Yaskawa INFORM job: DEMO_ROOF_SIDE_0625_3PAINT_12.JBI

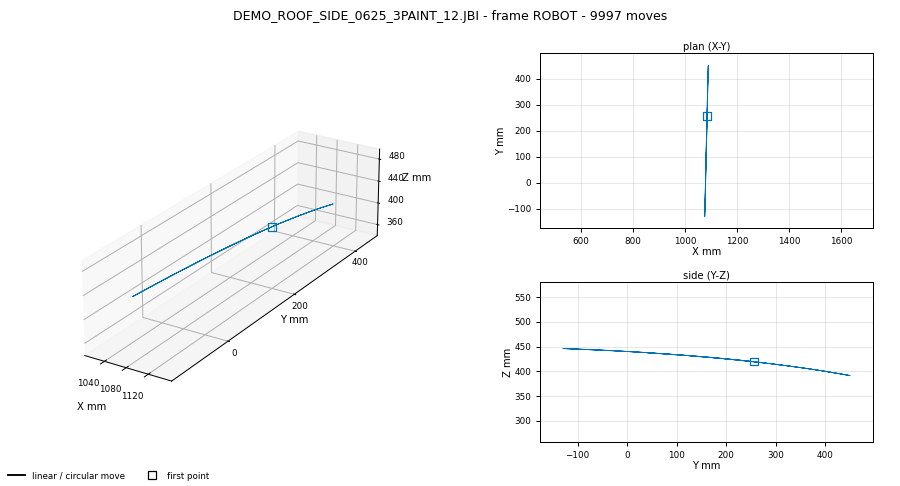
[picture p0: tool path of DEMO_ROOF_SIDE_0625_3PAINT_12.JBI in frame ROBOT, 9997 of 9997 moves have a stored position in this frame; points joined in program order, loops and branches not executed]
/JOB
//NAME DEMO_ROOF_SIDE_0625_3PAINT12
//POS
///NPOS 9997,0,0,0,0,0
///TOOL 0
///USER 0
///POSTYPE ROBOT
///RECTAN
///RCONF 1,0,0,0,0,0,0,0,0,0,0,0,0,0,0,0,0,0,0,0,0,0,0,0
C00000=1085.651,255.676,419.931,175.989,23.066,153.710
C00001=1085.645,255.428,419.959,175.986,23.063,153.710
C00002=1085.640,255.179,419.986,175.983,23.060,153.710
C00003=1085.635,254.931,420.014,175.981,23.057,153.709
C00004=1085.628,254.682,420.041,175.978,23.054,153.709
C00005=1085.623,254.434,420.069,175.975,23.051,153.709
C00006=1085.617,254.186,420.096,175.973,23.048,153.709
C00007=1085.611,253.937,420.124,175.970,23.045,153.708
C00008=1085.606,253.689,420.151,175.967,23.041,153.708
C00009=1085.600,253.441,420.179,175.965,23.039,153.708
C00010=1085.595,253.192,420.206,175.962,23.035,153.707
C00011=1085.589,252.943,420.233,175.959,23.032,153.707
C00012=1085.584,252.695,420.261,175.956,23.029,153.707
C00013=1085.578,252.446,420.287,175.953,23.026,153.707
C00014=1085.573,252.198,420.315,175.951,23.024,153.706
C00015=1085.567,251.950,420.342,175.948,23.020,153.706
C00016=1085.561,251.701,420.370,175.945,23.017,153.706
C00017=1085.555,251.453,420.397,175.943,23.014,153.705
C00018=1085.550,251.204,420.424,175.940,23.011,153.705
C00019=1085.544,250.956,420.451,175.937,23.008,153.705
C00020=1085.539,250.707,420.478,175.935,23.005,153.705
C00021=1085.532,250.459,420.506,175.932,23.002,153.704
C00022=1085.527,250.210,420.533,175.929,22.999,153.704
C00023=1085.519,249.831,420.575,175.925,22.995,153.704
C00024=1085.511,249.453,420.616,175.921,22.990,153.703
C00025=1085.502,249.074,420.657,175.917,22.986,153.703
C00026=1085.494,248.695,420.698,175.912,22.980,153.702
C00027=1085.488,248.447,420.725,175.910,22.978,153.702
C00028=1085.483,248.199,420.753,175.907,22.974,153.702
C00029=1085.477,247.950,420.780,175.905,22.972,153.702
C00030=1085.471,247.702,420.806,175.902,22.969,153.701
C00031=1085.466,247.453,420.834,175.899,22.965,153.701
C00032=1085.460,247.204,420.861,175.897,22.963,153.701
C00033=1085.455,246.956,420.888,175.894,22.959,153.700
C00034=1085.449,246.707,420.915,175.892,22.957,153.700
C00035=1085.443,246.459,420.941,175.889,22.954,153.700
C00036=1085.438,246.210,420.968,175.886,22.951,153.700
C00037=1085.432,245.962,420.995,175.883,22.948,153.699
C00038=1085.427,245.713,421.022,175.880,22.945,153.699
C00039=1085.421,245.465,421.048,175.878,22.942,153.699
C00040=1085.416,245.216,421.076,175.875,22.939,153.699
C00041=1085.409,244.967,421.103,175.872,22.936,153.698
C00042=1085.404,244.719,421.129,175.870,22.933,153.698
C00043=1085.398,244.471,421.156,175.867,22.930,153.698
C00044=1085.393,244.222,421.183,175.865,22.927,153.698
C00045=1085.387,243.974,421.210,175.862,22.924,153.697
C00046=1085.381,243.725,421.236,175.859,22.921,153.697
C00047=1085.376,243.477,421.263,175.857,22.918,153.697
C00048=1085.370,243.228,421.290,175.854,22.915,153.696
C00049=1085.365,242.980,421.317,175.851,22.912,153.696
C00050=1085.359,242.731,421.343,175.848,22.909,153.696
C00051=1085.353,242.482,421.370,175.845,22.906,153.696
C00052=1085.348,242.234,421.396,175.843,22.903,153.695
C00053=1085.342,241.986,421.423,175.840,22.900,153.695
C00054=1085.336,241.737,421.450,175.838,22.897,153.695
C00055=1085.330,241.489,421.476,175.835,22.894,153.695
C00056=1085.325,241.240,421.502,175.833,22.892,153.694
C00057=1085.319,240.992,421.529,175.830,22.889,153.694
C00058=1085.313,240.743,421.556,175.827,22.885,153.694
C00059=1085.307,240.494,421.582,175.824,22.883,153.694
C00060=1085.302,240.245,421.608,175.821,22.880,153.693
C00061=1085.296,239.997,421.635,175.819,22.877,153.693
C00062=1085.291,239.748,421.662,175.816,22.874,153.693
C00063=1085.285,239.500,421.688,175.814,22.871,153.693
C00064=1085.279,239.251,421.714,175.811,22.868,153.692
C00065=1085.273,239.003,421.741,175.809,22.865,153.692
C00066=1085.267,238.754,421.767,175.806,22.863,153.692
C00067=1085.262,238.506,421.793,175.803,22.859,153.692
C00068=1085.257,238.258,421.820,175.800,22.857,153.691
C00069=1085.251,238.009,421.846,175.797,22.853,153.691
C00070=1085.245,237.761,421.872,175.795,22.851,153.691
C00071=1085.240,237.512,421.898,175.792,22.848,153.691
C00072=1085.234,237.263,421.925,175.790,22.845,153.690
C00073=1085.228,237.015,421.952,175.787,22.842,153.690
C00074=1085.223,236.766,421.977,175.785,22.839,153.690
C00075=1085.214,236.380,422.019,175.780,22.834,153.690
C00076=1085.205,235.995,422.059,175.777,22.830,153.689
C00077=1085.196,235.609,422.100,175.772,22.825,153.689
C00078=1085.188,235.224,422.140,175.768,22.821,153.688
C00079=1085.182,234.975,422.166,175.765,22.818,153.688
C00080=1085.177,234.726,422.192,175.763,22.815,153.688
C00081=1085.171,234.478,422.219,175.760,22.812,153.688
C00082=1085.165,234.229,422.244,175.758,22.809,153.687
C00083=1085.159,233.981,422.271,175.755,22.806,153.687
C00084=1085.154,233.732,422.297,175.753,22.804,153.687
C00085=1085.149,233.484,422.323,175.750,22.800,153.687
C00086=1085.143,233.235,422.349,175.748,22.798,153.686
C00087=1085.138,232.986,422.375,175.745,22.794,153.686
C00088=1085.131,232.738,422.400,175.742,22.791,153.686
C00089=1085.126,232.489,422.427,175.739,22.789,153.686
C00090=1085.120,232.240,422.453,175.736,22.786,153.685
C00091=1085.115,231.991,422.479,175.734,22.783,153.685
C00092=1085.109,231.744,422.505,175.731,22.780,153.685
C00093=1085.103,231.495,422.531,175.729,22.777,153.684
C00094=1085.098,231.246,422.557,175.726,22.774,153.684
C00095=1085.092,230.997,422.582,175.724,22.771,153.684
C00096=1085.086,230.749,422.609,175.721,22.768,153.684
C00097=1085.081,230.501,422.634,175.719,22.765,153.683
C00098=1085.076,230.252,422.660,175.716,22.762,153.683
C00099=1085.069,230.003,422.685,175.713,22.760,153.683
C00100=1085.064,229.754,422.711,175.710,22.757,153.683
C00101=1085.058,229.506,422.738,175.708,22.754,153.682
C00102=1085.052,229.257,422.763,175.705,22.751,153.682
C00103=1085.047,229.009,422.789,175.703,22.748,153.682
C00104=1085.041,228.760,422.814,175.700,22.745,153.682
C00105=1085.035,228.511,422.840,175.698,22.742,153.681
C00106=1085.030,228.262,422.866,175.696,22.740,153.681
C00107=1085.024,228.013,422.891,175.692,22.737,153.681
C00108=1085.019,227.765,422.917,175.690,22.734,153.681
C00109=1085.013,227.516,422.942,175.687,22.731,153.681
C00110=1085.007,227.267,422.968,175.685,22.728,153.680
C00111=1085.001,227.019,422.994,175.682,22.725,153.680
C00112=1084.996,226.771,423.020,175.680,22.722,153.680
C00113=1084.990,226.522,423.045,175.677,22.719,153.680
C00114=1084.984,226.273,423.071,175.675,22.716,153.679
C00115=1084.979,226.024,423.097,175.672,22.714,153.679
C00116=1084.973,225.777,423.122,175.669,22.711,153.679
C00117=1084.968,225.528,423.148,175.666,22.708,153.679
C00118=1084.962,225.278,423.173,175.664,22.705,153.678
C00119=1084.957,225.030,423.198,175.661,22.702,153.678
C00120=1084.951,224.781,423.223,175.659,22.699,153.678
C00121=1084.945,224.532,423.249,175.656,22.696,153.678
C00122=1084.939,224.284,423.275,175.654,22.693,153.677
C00123=1084.934,224.035,423.300,175.652,22.691,153.677
C00124=1084.928,223.787,423.326,175.649,22.688,153.677
C00125=1084.923,223.538,423.351,175.646,22.685,153.677
C00126=1084.917,223.290,423.377,175.643,22.682,153.676
C00127=1084.908,222.895,423.417,175.640,22.678,153.676
C00128=1084.900,222.501,423.457,175.635,22.673,153.675
C00129=1084.890,222.107,423.497,175.632,22.668,153.675
C00130=1084.882,221.713,423.537,175.627,22.663,153.675
C00131=1084.875,221.464,423.562,175.625,22.661,153.675
C00132=1084.870,221.215,423.588,175.622,22.658,153.674
C00133=1084.865,220.967,423.612,175.620,22.655,153.674
C00134=1084.858,220.718,423.637,175.618,22.652,153.674
C00135=1084.853,220.469,423.663,175.615,22.649,153.674
C00136=1084.847,220.221,423.688,175.612,22.647,153.673
C00137=1084.841,219.972,423.713,175.609,22.643,153.673
C00138=1084.836,219.724,423.738,175.607,22.641,153.673
C00139=1084.830,219.475,423.764,175.604,22.638,153.673
C00140=1084.824,219.226,423.789,175.602,22.635,153.672
C00141=1084.819,218.978,423.813,175.600,22.632,153.672
C00142=1084.813,218.729,423.839,175.597,22.630,153.672
C00143=1084.808,218.480,423.864,175.595,22.627,153.672
C00144=1084.802,218.231,423.889,175.592,22.623,153.671
C00145=1084.796,217.982,423.914,175.590,22.621,153.671
C00146=1084.790,217.734,423.939,175.586,22.618,153.671
C00147=1084.784,217.485,423.963,175.584,22.615,153.671
C00148=1084.780,217.237,423.989,175.582,22.612,153.670
C00149=1084.773,216.988,424.014,175.579,22.609,153.670
C00150=1084.768,216.739,424.038,175.577,22.607,153.670
C00151=1084.762,216.491,424.064,175.574,22.604,153.670
C00152=1084.757,216.242,424.088,175.572,22.601,153.669
C00153=1084.751,215.993,424.114,175.570,22.598,153.669
C00154=1084.746,215.745,424.138,175.566,22.595,153.669
C00155=1084.740,215.496,424.164,175.564,22.592,153.669
C00156=1084.734,215.247,424.188,175.561,22.589,153.668
C00157=1084.728,214.998,424.212,175.559,22.586,153.668
C00158=1084.724,214.750,424.238,175.557,22.584,153.668
C00159=1084.718,214.500,424.263,175.554,22.581,153.668
C00160=1084.712,214.252,424.288,175.552,22.578,153.667
C00161=1084.706,214.003,424.312,175.549,22.575,153.667
C00162=1084.701,213.755,424.336,175.547,22.572,153.667
C00163=1084.695,213.506,424.362,175.544,22.570,153.667
C00164=1084.689,213.257,424.386,175.541,22.566,153.666
C00165=1084.683,213.009,424.411,175.539,22.564,153.666
C00166=1084.679,212.760,424.436,175.536,22.560,153.666
C00167=1084.673,212.510,424.461,175.534,22.558,153.666
C00168=1084.667,212.262,424.485,175.532,22.555,153.665
C00169=1084.661,212.013,424.510,175.529,22.552,153.665
C00170=1084.656,211.765,424.535,175.527,22.549,153.665
C00171=1084.651,211.516,424.559,175.524,22.546,153.665
C00172=1084.644,211.267,424.584,175.522,22.544,153.664
C00173=1084.639,211.019,424.609,175.520,22.541,153.664
C00174=1084.633,210.770,424.633,175.517,22.538,153.664
C00175=1084.628,210.521,424.657,175.514,22.535,153.664
C00176=1084.622,210.272,424.682,175.512,22.532,153.663
C00177=1084.616,210.024,424.706,175.509,22.529,153.663
C00178=1084.610,209.775,424.731,175.507,22.526,153.663
C00179=1084.602,209.385,424.769,175.503,22.522,153.663
C00180=1084.592,208.995,424.808,175.499,22.518,153.662
C00181=1084.584,208.604,424.846,175.495,22.513,153.662
C00182=1084.575,208.214,424.884,175.492,22.509,153.661
C00183=1084.552,207.186,424.984,175.406,22.464,153.664
C00184=1084.547,206.937,425.007,175.403,22.462,153.664
C00185=1084.540,206.688,425.031,175.401,22.460,153.664
C00186=1084.535,206.439,425.056,175.398,22.458,153.664
C00187=1084.530,206.190,425.080,175.396,22.457,153.664
C00188=1084.524,205.941,425.103,175.393,22.455,153.664
C00189=1084.519,205.693,425.127,175.391,22.453,153.664
C00190=1084.512,205.444,425.151,175.387,22.451,153.664
C00191=1084.507,205.195,425.175,175.385,22.448,153.664
C00192=1084.502,204.946,425.199,175.383,22.447,153.664
C00193=1084.496,204.698,425.222,175.380,22.445,153.664
C00194=1084.491,204.449,425.246,175.378,22.443,153.664
C00195=1084.485,204.200,425.270,175.375,22.441,153.664
C00196=1084.479,203.952,425.294,175.373,22.439,153.664
C00197=1084.474,203.702,425.318,175.370,22.437,153.664
C00198=1084.468,203.454,425.342,175.367,22.435,153.664
C00199=1084.463,203.204,425.365,175.365,22.433,153.664
C00200=1084.457,202.956,425.389,175.362,22.431,153.664
C00201=1084.452,202.707,425.412,175.360,22.429,153.664
C00202=1084.446,202.458,425.437,175.357,22.428,153.664
C00203=1084.441,202.209,425.459,175.355,22.426,153.664
C00204=1084.434,201.960,425.483,175.352,22.424,153.664
C00205=1084.429,201.711,425.507,175.349,22.422,153.664
C00206=1084.423,201.463,425.531,175.347,22.420,153.664
C00207=1084.418,201.214,425.554,175.344,22.418,153.664
C00208=1084.412,200.965,425.578,175.342,22.416,153.664
C00209=1084.406,200.717,425.601,175.339,22.414,153.664
C00210=1084.401,200.468,425.625,175.337,22.413,153.664
C00211=1084.395,200.218,425.648,175.334,22.411,153.664
C00212=1084.389,199.970,425.672,175.332,22.409,153.664
C00213=1084.384,199.721,425.696,175.329,22.407,153.664
C00214=1084.378,199.473,425.719,175.327,22.405,153.664
C00215=1084.372,199.224,425.742,175.323,22.403,153.664
C00216=1084.367,198.974,425.766,175.321,22.401,153.664
C00217=1084.361,198.726,425.789,175.319,22.400,153.664
C00218=1084.355,198.477,425.812,175.316,22.398,153.664
C00219=1084.350,198.228,425.836,175.314,22.396,153.664
C00220=1084.344,197.980,425.860,175.311,22.394,153.664
C00221=1084.338,197.731,425.882,175.309,22.392,153.664
C00222=1084.333,197.481,425.906,175.306,22.390,153.663
C00223=1084.327,197.233,425.930,175.304,22.389,153.663
C00224=1084.321,196.984,425.953,175.301,22.387,153.663
C00225=1084.316,196.735,425.977,175.299,22.385,153.663
C00226=1084.310,196.486,426.000,175.296,22.383,153.663
C00227=1084.304,196.237,426.023,175.293,22.381,153.663
C00228=1084.299,195.988,426.047,175.291,22.379,153.663
C00229=1084.293,195.739,426.070,175.288,22.377,153.663
C00230=1084.287,195.491,426.093,175.286,22.375,153.663
C00231=1084.282,195.242,426.116,175.283,22.373,153.663
C00232=1084.277,194.993,426.140,175.281,22.371,153.663
C00233=1084.271,194.744,426.163,175.278,22.370,153.663
C00234=1084.265,194.495,426.186,175.276,22.368,153.663
C00235=1084.259,194.247,426.209,175.273,22.366,153.663
C00236=1084.254,193.998,426.233,175.271,22.364,153.663
C00237=1084.248,193.749,426.256,175.268,22.362,153.663
C00238=1084.243,193.500,426.279,175.266,22.361,153.663
C00239=1084.237,193.251,426.302,175.264,22.359,153.663
C00240=1084.232,193.002,426.325,175.261,22.356,153.663
C00241=1084.226,192.753,426.348,175.259,22.355,153.663
C00242=1084.221,192.505,426.371,175.256,22.353,153.663
C00243=1084.215,192.256,426.394,175.254,22.351,153.663
C00244=1084.209,191.977,426.420,175.251,22.349,153.663
C00245=1084.203,191.699,426.446,175.248,22.347,153.663
C00246=1084.197,191.420,426.472,175.245,22.344,153.663
C00247=1084.190,191.142,426.498,175.242,22.342,153.663
C00248=1084.185,190.893,426.521,175.240,22.341,153.663
C00249=1084.180,190.644,426.544,175.238,22.339,153.663
C00250=1084.174,190.395,426.567,175.235,22.337,153.663
C00251=1084.168,190.146,426.590,175.233,22.335,153.663
C00252=1084.162,189.897,426.613,175.230,22.333,153.663
C00253=1084.157,189.648,426.636,175.228,22.331,153.663
C00254=1084.152,189.400,426.659,175.225,22.329,153.663
C00255=1084.147,189.151,426.682,175.223,22.327,153.662
C00256=1084.141,188.902,426.705,175.220,22.326,153.662
C00257=1084.135,188.653,426.728,175.218,22.323,153.662
C00258=1084.129,188.404,426.751,175.216,22.321,153.662
C00259=1084.125,188.154,426.774,175.213,22.320,153.662
C00260=1084.120,187.906,426.796,175.211,22.318,153.662
C00261=1084.114,187.657,426.819,175.208,22.316,153.662
C00262=1084.108,187.408,426.842,175.206,22.314,153.662
C00263=1084.102,187.159,426.865,175.204,22.312,153.662
C00264=1084.097,186.910,426.888,175.201,22.310,153.662
C00265=1084.092,186.662,426.911,175.199,22.308,153.662
C00266=1084.087,186.412,426.933,175.196,22.306,153.662
C00267=1084.081,186.163,426.956,175.194,22.304,153.662
C00268=1084.075,185.915,426.979,175.191,22.302,153.662
C00269=1084.070,185.666,427.002,175.189,22.300,153.662
C00270=1084.065,185.418,427.025,175.187,22.299,153.662
C00271=1084.059,185.168,427.047,175.184,22.296,153.662
C00272=1084.053,184.919,427.070,175.182,22.295,153.662
C00273=1084.048,184.670,427.093,175.179,22.293,153.662
C00274=1084.042,184.421,427.116,175.177,22.291,153.662
C00275=1084.036,184.172,427.138,175.174,22.289,153.662
C00276=1084.031,183.924,427.160,175.172,22.287,153.662
C00277=1084.025,183.675,427.183,175.169,22.285,153.662
C00278=1084.019,183.426,427.206,175.167,22.284,153.662
C00279=1084.014,183.177,427.228,175.165,22.282,153.662
C00280=1084.007,182.928,427.251,175.162,22.280,153.662
C00281=1084.002,182.679,427.274,175.160,22.278,153.662
C00282=1083.996,182.430,427.296,175.157,22.276,153.662
C00283=1083.991,182.181,427.318,175.155,22.275,153.662
C00284=1083.985,181.933,427.341,175.152,22.273,153.661
C00285=1083.979,181.683,427.363,175.150,22.271,153.661
C00286=1083.973,181.434,427.386,175.147,22.269,153.661
C00287=1083.967,181.185,427.408,175.145,22.267,153.661
C00288=1083.961,180.936,427.430,175.142,22.265,153.661
C00289=1083.956,180.688,427.453,175.141,22.264,153.661
C00290=1083.951,180.439,427.475,175.138,22.262,153.661
C00291=1083.944,180.190,427.498,175.136,22.260,153.661
C00292=1083.939,179.940,427.520,175.133,22.259,153.661
C00293=1083.933,179.692,427.543,175.131,22.257,153.661
C00294=1083.928,179.443,427.564,175.129,22.254,153.661
C00295=1083.922,179.194,427.587,175.126,22.253,153.661
C00296=1083.917,178.945,427.609,175.124,22.251,153.661
C00297=1083.910,178.696,427.632,175.121,22.249,153.661
C00298=1083.905,178.447,427.653,175.119,22.247,153.661
C00299=1083.900,178.198,427.676,175.116,22.245,153.661
C00300=1083.893,177.949,427.698,175.114,22.244,153.661
C00301=1083.888,177.700,427.721,175.111,22.242,153.661
C00302=1083.883,177.451,427.743,175.109,22.240,153.661
C00303=1083.876,177.203,427.765,175.106,22.238,153.661
C00304=1083.871,176.953,427.787,175.105,22.236,153.661
C00305=1083.866,176.705,427.809,175.103,22.234,153.661
C00306=1083.860,176.456,427.832,175.100,22.233,153.661
C00307=1083.854,176.206,427.854,175.098,22.231,153.661
C00308=1083.848,175.928,427.879,175.095,22.229,153.661
C00309=1083.841,175.649,427.904,175.092,22.226,153.661
C00310=1083.836,175.370,427.929,175.090,22.224,153.661
C00311=1083.830,175.091,427.953,175.087,22.223,153.661
C00312=1083.823,174.842,427.975,175.085,22.221,153.661
C00313=1083.818,174.593,427.998,175.082,22.218,153.661
C00314=1083.813,174.344,428.020,175.080,22.217,153.660
C00315=1083.807,174.095,428.041,175.078,22.215,153.660
C00316=1083.801,173.846,428.064,175.075,22.213,153.660
C00317=1083.795,173.598,428.086,175.073,22.211,153.660
C00318=1083.790,173.348,428.108,175.070,22.209,153.660
C00319=1083.785,173.099,428.130,175.069,22.207,153.660
C00320=1083.779,172.851,428.152,175.066,22.206,153.660
C00321=1083.773,172.601,428.174,175.064,22.204,153.660
C00322=1083.768,172.353,428.196,175.061,22.202,153.660
C00323=1083.762,172.103,428.218,175.059,22.200,153.660
C00324=1083.757,171.854,428.240,175.057,22.198,153.660
C00325=1083.751,171.606,428.262,175.054,22.196,153.660
C00326=1083.745,171.356,428.284,175.052,22.194,153.660
C00327=1083.740,171.108,428.306,175.049,22.192,153.660
C00328=1083.735,170.858,428.328,175.048,22.190,153.660
C00329=1083.729,170.610,428.349,175.045,22.189,153.660
C00330=1083.724,170.360,428.371,175.043,22.187,153.660
C00331=1083.717,170.112,428.394,175.041,22.185,153.660
C00332=1083.712,169.863,428.415,175.038,22.183,153.660
C00333=1083.706,169.614,428.437,175.036,22.181,153.660
C00334=1083.701,169.365,428.459,175.033,22.179,153.660
C00335=1083.696,169.115,428.481,175.031,22.177,153.659
C00336=1083.690,168.867,428.502,175.029,22.175,153.659
C00337=1083.685,168.617,428.525,175.027,22.174,153.659
C00338=1083.679,168.369,428.546,175.025,22.172,153.659
C00339=1083.674,168.119,428.568,175.022,22.169,153.659
C00340=1083.668,167.871,428.589,175.020,22.168,153.659
C00341=1083.663,167.621,428.612,175.017,22.166,153.659
C00342=1083.657,167.373,428.633,175.015,22.163,153.659
C00343=1083.652,167.123,428.655,175.014,22.162,153.659
C00344=1083.646,166.875,428.676,175.011,22.160,153.659
C00345=1083.641,166.625,428.699,175.009,22.158,153.659
C00346=1083.635,166.377,428.720,175.006,22.156,153.659
C00347=1083.630,166.127,428.742,175.004,22.154,153.659
C00348=1083.624,165.879,428.763,175.002,22.152,153.659
C00349=1083.620,165.630,428.785,174.999,22.150,153.659
C00350=1083.613,165.381,428.807,174.998,22.149,153.659
C00351=1083.609,165.132,428.829,174.995,22.146,153.658
C00352=1083.602,164.883,428.850,174.993,22.145,153.658
C00353=1083.597,164.634,428.872,174.990,22.143,153.658
C00354=1083.591,164.385,428.894,174.988,22.140,153.658
C00355=1083.586,164.136,428.915,174.986,22.139,153.658
C00356=1083.581,163.887,428.937,174.984,22.137,153.658
C00357=1083.575,163.638,428.959,174.982,22.135,153.658
C00358=1083.570,163.389,428.980,174.979,22.133,153.658
C00359=1083.564,163.140,429.002,174.977,22.131,153.658
C00360=1083.559,162.891,429.023,174.975,22.129,153.658
C00361=1083.554,162.642,429.045,174.972,22.127,153.658
C00362=1083.548,162.393,429.066,174.971,22.125,153.658
C00363=1083.543,162.144,429.088,174.968,22.123,153.658
C00364=1083.538,161.895,429.109,174.966,22.121,153.658
C00365=1083.532,161.646,429.131,174.964,22.119,153.658
C00366=1083.527,161.397,429.152,174.961,22.117,153.657
C00367=1083.520,161.148,429.174,174.959,22.115,153.657
C00368=1083.515,160.899,429.194,174.957,22.114,153.657
C00369=1083.509,160.650,429.216,174.955,22.112,153.657
C00370=1083.504,160.401,429.238,174.953,22.109,153.657
C00371=1083.499,160.152,429.259,174.950,22.108,153.657
C00372=1083.492,159.872,429.283,174.948,22.106,153.657
C00373=1083.486,159.593,429.306,174.945,22.103,153.657
C00374=1083.480,159.314,429.330,174.943,22.102,153.657
C00375=1083.473,159.034,429.355,174.941,22.099,153.657
C00376=1083.468,158.785,429.375,174.938,22.097,153.657
C00377=1083.462,158.537,429.397,174.936,22.096,153.657
C00378=1083.456,158.288,429.418,174.934,22.093,153.657
C00379=1083.451,158.038,429.439,174.931,22.091,153.657
C00380=1083.445,157.789,429.461,174.930,22.090,153.657
C00381=1083.439,157.541,429.482,174.927,22.088,153.657
C00382=1083.435,157.291,429.503,174.925,22.086,153.657
C00383=1083.428,157.042,429.525,174.922,22.084,153.657
C00384=1083.423,156.793,429.545,174.920,22.082,153.656
C00385=1083.418,156.545,429.566,174.919,22.080,153.656
C00386=1083.411,156.295,429.588,174.916,22.079,153.656
C00387=1083.406,156.046,429.609,174.914,22.076,153.656
C00388=1083.401,155.798,429.630,174.911,22.074,153.656
C00389=1083.395,155.548,429.651,174.910,22.072,153.656
C00390=1083.389,155.299,429.672,174.908,22.071,153.656
C00391=1083.383,155.050,429.693,174.905,22.069,153.656
C00392=1083.378,154.801,429.714,174.903,22.066,153.656
C00393=1083.372,154.552,429.735,174.900,22.065,153.656
C00394=1083.366,154.303,429.756,174.899,22.063,153.656
C00395=1083.361,154.054,429.777,174.897,22.061,153.656
C00396=1083.355,153.805,429.798,174.894,22.059,153.656
C00397=1083.350,153.556,429.819,174.892,22.057,153.656
C00398=1083.344,153.307,429.840,174.890,22.055,153.655
C00399=1083.339,153.058,429.861,174.888,22.054,153.655
C00400=1083.333,152.809,429.882,174.885,22.052,153.655
C00401=1083.327,152.559,429.903,174.883,22.049,153.655
C00402=1083.322,152.310,429.924,174.882,22.048,153.655
C00403=1083.317,152.062,429.945,174.879,22.046,153.655
C00404=1083.311,151.812,429.966,174.877,22.044,153.655
C00405=1083.305,151.563,429.987,174.874,22.042,153.655
C00406=1083.300,151.314,430.008,174.873,22.040,153.655
C00407=1083.295,151.065,430.028,174.871,22.038,153.655
C00408=1083.288,150.816,430.050,174.868,22.036,153.655
C00409=1083.282,150.567,430.070,174.866,22.034,153.655
C00410=1083.277,150.318,430.090,174.864,22.033,153.655
C00411=1083.272,150.069,430.112,174.862,22.030,153.655
C00412=1083.266,149.820,430.133,174.860,22.029,153.654
C00413=1083.261,149.570,430.153,174.857,22.026,153.654
C00414=1083.255,149.322,430.175,174.856,22.025,153.654
C00415=1083.250,149.073,430.195,174.853,22.022,153.654
C00416=1083.244,148.823,430.216,174.851,22.021,153.654
C00417=1083.238,148.574,430.236,174.849,22.019,153.654
C00418=1083.232,148.326,430.257,174.847,22.017,153.654
C00419=1083.227,148.077,430.278,174.845,22.015,153.654
C00420=1083.221,147.827,430.299,174.842,22.013,153.654
C00421=1083.216,147.578,430.319,174.840,22.011,153.654
C00422=1083.210,147.329,430.340,174.838,22.010,153.654
C00423=1083.204,147.080,430.360,174.836,22.007,153.654
C00424=1083.199,146.830,430.381,174.834,22.005,153.654
C00425=1083.193,146.581,430.402,174.832,22.003,153.653
C00426=1083.187,146.333,430.422,174.830,22.002,153.653
C00427=1083.182,146.083,430.442,174.827,22.000,153.653
C00428=1083.176,145.835,430.464,174.825,21.997,153.653
C00429=1083.171,145.585,430.485,174.824,21.996,153.653
C00430=1083.165,145.336,430.505,174.821,21.994,153.653
C00431=1083.159,145.087,430.525,174.819,21.992,153.653
C00432=1083.154,144.838,430.546,174.817,21.990,153.653
C00433=1083.148,144.589,430.566,174.815,21.988,153.653
C00434=1083.142,144.339,430.587,174.813,21.986,153.653
C00435=1083.137,144.090,430.607,174.810,21.984,153.653
C00436=1083.131,143.811,430.630,174.808,21.982,153.653
C00437=1083.124,143.532,430.653,174.806,21.980,153.653
C00438=1083.119,143.252,430.676,174.803,21.977,153.652
C00439=1083.112,142.973,430.699,174.801,21.975,153.652
C00440=1083.107,142.724,430.719,174.799,21.973,153.652
C00441=1083.100,142.474,430.740,174.797,21.971,153.652
C00442=1083.095,142.225,430.760,174.795,21.970,153.652
C00443=1083.089,141.976,430.782,174.793,21.967,153.652
C00444=1083.083,141.728,430.802,174.791,21.966,153.652
C00445=1083.078,141.478,430.821,174.789,21.963,153.652
C00446=1083.073,141.229,430.842,174.786,21.962,153.652
C00447=1083.067,140.980,430.862,174.785,21.960,153.652
C00448=1083.062,140.731,430.882,174.783,21.958,153.652
C00449=1083.056,140.482,430.902,174.780,21.956,153.651
C00450=1083.050,140.232,430.923,174.779,21.954,153.651
C00451=1083.045,139.983,430.944,174.776,21.952,153.651
C00452=1083.039,139.734,430.964,174.774,21.950,153.651
C00453=1083.034,139.485,430.984,174.772,21.948,153.651
C00454=1083.028,139.236,431.004,174.770,21.946,153.651
C00455=1083.022,138.987,431.025,174.768,21.944,153.651
C00456=1083.016,138.738,431.045,174.766,21.942,153.651
C00457=1083.011,138.489,431.065,174.764,21.940,153.651
C00458=1083.005,138.240,431.085,174.762,21.938,153.651
C00459=1083.000,137.991,431.105,174.759,21.936,153.651
C00460=1082.994,137.741,431.125,174.758,21.935,153.651
C00461=1082.988,137.492,431.146,174.756,21.932,153.650
C00462=1082.982,137.243,431.166,174.753,21.930,153.650
C00463=1082.977,136.994,431.187,174.752,21.928,153.650
C00464=1082.971,136.745,431.206,174.750,21.926,153.650
C00465=1082.966,136.496,431.226,174.747,21.924,153.650
C00466=1082.960,136.247,431.246,174.746,21.922,153.650
C00467=1082.954,135.998,431.266,174.743,21.921,153.650
C00468=1082.949,135.749,431.287,174.741,21.918,153.650
C00469=1082.943,135.499,431.306,174.739,21.917,153.650
C00470=1082.938,135.250,431.327,174.737,21.914,153.650
C00471=1082.932,135.001,431.347,174.735,21.913,153.650
C00472=1082.927,134.752,431.367,174.733,21.911,153.649
C00473=1082.921,134.503,431.386,174.731,21.908,153.649
C00474=1082.916,134.254,431.407,174.729,21.906,153.649
C00475=1082.910,134.005,431.427,174.727,21.905,153.649
C00476=1082.904,133.755,431.446,174.725,21.903,153.649
C00477=1082.899,133.506,431.467,174.723,21.900,153.649
C00478=1082.893,133.258,431.487,174.721,21.898,153.649
C00479=1082.888,133.008,431.506,174.719,21.897,153.649
C00480=1082.882,132.759,431.526,174.717,21.894,153.649
C00481=1082.876,132.510,431.546,174.715,21.893,153.649
C00482=1082.871,132.260,431.566,174.713,21.891,153.648
C00483=1082.865,132.012,431.586,174.711,21.888,153.648
C00484=1082.859,131.763,431.606,174.709,21.887,153.648
C00485=1082.853,131.513,431.625,174.707,21.884,153.648
C00486=1082.848,131.264,431.646,174.705,21.883,153.648
C00487=1082.842,131.015,431.665,174.703,21.881,153.648
C00488=1082.836,130.766,431.685,174.700,21.879,153.648
C00489=1082.830,130.517,431.705,174.699,21.877,153.648
C00490=1082.825,130.268,431.724,174.697,21.875,153.648
C00491=1082.819,130.019,431.745,174.694,21.873,153.648
C00492=1082.814,129.769,431.764,174.693,21.871,153.647
C00493=1082.808,129.520,431.784,174.691,21.869,153.647
C00494=1082.802,129.271,431.803,174.688,21.867,153.647
C00495=1082.796,129.022,431.823,174.687,21.865,153.647
C00496=1082.790,128.773,431.843,174.685,21.863,153.647
C00497=1082.785,128.524,431.863,174.683,21.861,153.647
C00498=1082.779,128.274,431.882,174.681,21.859,153.647
C00499=1082.773,128.025,431.902,174.678,21.857,153.647
C00500=1082.767,127.745,431.924,174.676,21.855,153.647
C00501=1082.760,127.466,431.946,174.674,21.853,153.647
C00502=1082.754,127.186,431.969,174.672,21.851,153.646
C00503=1082.748,126.906,431.991,174.670,21.848,153.646
C00504=1082.742,126.657,432.010,174.668,21.846,153.646
C00505=1082.736,126.408,432.030,174.665,21.844,153.646
C00506=1082.731,126.159,432.049,174.664,21.842,153.646
C00507=1082.725,125.909,432.068,174.662,21.840,153.646
C00508=1082.719,125.661,432.088,174.660,21.838,153.646
C00509=1082.713,125.411,432.108,174.658,21.837,153.646
C00510=1082.708,125.163,432.127,174.656,21.834,153.646
C00511=1082.703,124.913,432.147,174.654,21.832,153.645
C00512=1082.697,124.664,432.166,174.652,21.831,153.645
C00513=1082.691,124.415,432.186,174.650,21.828,153.645
C00514=1082.685,124.166,432.205,174.648,21.826,153.645
C00515=1082.680,123.916,432.225,174.646,21.824,153.645
C00516=1082.674,123.667,432.245,174.644,21.822,153.645
C00517=1082.668,123.418,432.264,174.642,21.820,153.645
C00518=1082.662,123.168,432.283,174.640,21.818,153.645
C00519=1082.657,122.920,432.302,174.638,21.816,153.645
C00520=1082.651,122.671,432.322,174.636,21.814,153.644
C00521=1082.646,122.422,432.341,174.635,21.812,153.644
C00522=1082.641,122.172,432.361,174.632,21.810,153.644
C00523=1082.635,121.923,432.381,174.630,21.808,153.644
C00524=1082.629,121.674,432.400,174.629,21.806,153.644
C00525=1082.624,121.425,432.419,174.626,21.804,153.644
C00526=1082.618,121.175,432.438,174.625,21.802,153.644
C00527=1082.613,120.926,432.458,174.623,21.800,153.644
C00528=1082.607,120.677,432.478,174.620,21.798,153.643
C00529=1082.601,120.428,432.497,174.619,21.796,153.643
C00530=1082.596,120.179,432.516,174.617,21.794,153.643
C00531=1082.590,119.930,432.535,174.615,21.792,153.643
C00532=1082.584,119.680,432.554,174.613,21.789,153.643
C00533=1082.578,119.431,432.574,174.612,21.788,153.643
C00534=1082.573,119.182,432.593,174.609,21.785,153.643
C00535=1082.568,118.933,432.612,174.607,21.783,153.643
C00536=1082.562,118.684,432.632,174.606,21.781,153.642
C00537=1082.556,118.434,432.651,174.603,21.779,153.642
C00538=1082.551,118.185,432.670,174.602,21.777,153.642
C00539=1082.546,117.936,432.689,174.600,21.775,153.642
C00540=1082.540,117.687,432.708,174.597,21.773,153.642
C00541=1082.534,117.437,432.727,174.596,21.771,153.642
C00542=1082.528,117.188,432.747,174.594,21.769,153.642
C00543=1082.523,116.940,432.766,174.592,21.767,153.642
C00544=1082.517,116.690,432.785,174.590,21.764,153.641
C00545=1082.512,116.441,432.805,174.589,21.762,153.641
C00546=1082.507,116.192,432.824,174.586,21.761,153.641
C00547=1082.501,115.943,432.843,174.584,21.758,153.641
C00548=1082.495,115.693,432.862,174.583,21.756,153.641
C00549=1082.490,115.444,432.881,174.580,21.754,153.641
C00550=1082.484,115.195,432.900,174.579,21.752,153.641
C00551=1082.479,114.946,432.919,174.577,21.750,153.640
C00552=1082.473,114.696,432.939,174.575,21.748,153.640
C00553=1082.468,114.447,432.958,174.573,21.745,153.640
C00554=1082.462,114.198,432.977,174.572,21.744,153.640
C00555=1082.456,113.949,432.995,174.569,21.742,153.640
C00556=1082.450,113.699,433.015,174.567,21.739,153.640
C00557=1082.445,113.451,433.034,174.566,21.737,153.640
C00558=1082.440,113.201,433.052,174.564,21.735,153.640
C00559=1082.434,112.951,433.071,174.562,21.734,153.639
C00560=1082.428,112.703,433.090,174.560,21.731,153.639
C00561=1082.423,112.453,433.109,174.558,21.729,153.639
C00562=1082.417,112.204,433.128,174.556,21.727,153.639
C00563=1082.411,111.955,433.147,174.555,21.725,153.639
C00564=1082.405,111.676,433.168,174.553,21.723,153.639
C00565=1082.398,111.395,433.189,174.550,21.720,153.639
C00566=1082.392,111.116,433.210,174.548,21.718,153.638
C00567=1082.385,110.837,433.232,174.546,21.716,153.638
C00568=1082.380,110.587,433.250,174.544,21.714,153.638
C00569=1082.375,110.338,433.269,174.542,21.712,153.638
C00570=1082.368,110.089,433.288,174.541,21.710,153.638
C00571=1082.363,109.839,433.307,174.538,21.708,153.638
C00572=1082.357,109.590,433.326,174.536,21.705,153.638
C00573=1082.351,109.341,433.344,174.535,21.703,153.637
C00574=1082.346,109.092,433.363,174.533,21.701,153.637
C00575=1082.340,108.842,433.382,174.531,21.699,153.637
C00576=1082.334,108.594,433.401,174.529,21.697,153.637
C00577=1082.329,108.344,433.419,174.527,21.695,153.637
C00578=1082.322,108.095,433.438,174.525,21.693,153.637
C00579=1082.317,107.846,433.457,174.524,21.691,153.637
C00580=1082.312,107.596,433.476,174.522,21.689,153.637
C00581=1082.306,107.347,433.493,174.520,21.687,153.636
C00582=1082.300,107.098,433.513,174.518,21.685,153.636
C00583=1082.295,106.848,433.532,174.516,21.683,153.636
C00584=1082.289,106.599,433.550,174.514,21.680,153.636
C00585=1082.284,106.350,433.569,174.513,21.679,153.636
C00586=1082.277,106.101,433.587,174.511,21.676,153.636
C00587=1082.272,105.852,433.606,174.508,21.674,153.636
C00588=1082.267,105.602,433.625,174.507,21.672,153.635
C00589=1082.261,105.354,433.643,174.505,21.669,153.635
C00590=1082.255,105.104,433.662,174.503,21.668,153.635
C00591=1082.249,104.854,433.680,174.501,21.666,153.635
C00592=1082.244,104.606,433.699,174.500,21.664,153.635
C00593=1082.238,104.356,433.717,174.497,21.661,153.635
C00594=1082.233,104.107,433.736,174.496,21.659,153.635
C00595=1082.227,103.858,433.755,174.494,21.657,153.634
C00596=1082.221,103.608,433.773,174.492,21.655,153.634
C00597=1082.216,103.359,433.792,174.490,21.653,153.634
C00598=1082.210,103.110,433.810,174.489,21.651,153.634
C00599=1082.205,102.861,433.829,174.487,21.649,153.634
C00600=1082.199,102.611,433.847,174.485,21.647,153.634
C00601=1082.193,102.362,433.866,174.483,21.644,153.634
C00602=1082.187,102.113,433.884,174.482,21.642,153.633
C00603=1082.182,101.864,433.902,174.479,21.640,153.633
C00604=1082.177,101.614,433.921,174.478,21.638,153.633
C00605=1082.171,101.365,433.939,174.476,21.636,153.633
C00606=1082.166,101.115,433.958,174.475,21.634,153.633
C00607=1082.160,100.867,433.976,174.472,21.631,153.633
C00608=1082.154,100.617,433.994,174.471,21.629,153.632
C00609=1082.148,100.368,434.013,174.469,21.627,153.632
C00610=1082.143,100.119,434.031,174.467,21.625,153.632
C00611=1082.136,99.870,434.049,174.465,21.623,153.632
C00612=1082.131,99.620,434.068,174.464,21.621,153.632
C00613=1082.125,99.371,434.086,174.461,21.619,153.632
C00614=1082.119,99.122,434.104,174.460,21.617,153.632
C00615=1082.114,98.873,434.123,174.458,21.615,153.631
C00616=1082.108,98.624,434.141,174.456,21.613,153.631
C00617=1082.102,98.374,434.159,174.454,21.610,153.631
C00618=1082.096,98.125,434.178,174.453,21.608,153.631
C00619=1082.091,97.875,434.195,174.451,21.606,153.631
C00620=1082.085,97.626,434.213,174.449,21.604,153.631
C00621=1082.080,97.377,434.232,174.447,21.602,153.631
C00622=1082.074,97.127,434.250,174.446,21.600,153.630
C00623=1082.068,96.879,434.268,174.443,21.597,153.630
C00624=1082.062,96.629,434.287,174.442,21.596,153.630
C00625=1082.057,96.380,434.305,174.440,21.593,153.630
C00626=1082.050,96.131,434.323,174.438,21.591,153.630
C00627=1082.046,95.881,434.341,174.436,21.589,153.630
C00628=1082.039,95.602,434.361,174.435,21.587,153.629
C00629=1082.032,95.322,434.382,174.433,21.585,153.629
C00630=1082.026,95.042,434.402,174.431,21.582,153.629
C00631=1082.020,94.763,434.422,174.428,21.579,153.629
C00632=1082.015,94.514,434.440,174.427,21.577,153.629
C00633=1082.009,94.265,434.459,174.425,21.575,153.629
C00634=1082.003,94.015,434.476,174.423,21.573,153.628
C00635=1081.997,93.766,434.494,174.421,21.571,153.628
C00636=1081.992,93.516,434.513,174.420,21.569,153.628
C00637=1081.986,93.267,434.531,174.418,21.566,153.628
C00638=1081.980,93.018,434.549,174.416,21.564,153.628
C00639=1081.975,92.769,434.567,174.414,21.562,153.628
C00640=1081.969,92.519,434.585,174.413,21.560,153.627
C00641=1081.964,92.270,434.602,174.411,21.558,153.627
C00642=1081.957,92.021,434.621,174.409,21.556,153.627
C00643=1081.953,91.772,434.639,174.408,21.553,153.627
C00644=1081.947,91.523,434.657,174.406,21.551,153.627
C00645=1081.941,91.273,434.675,174.404,21.549,153.627
C00646=1081.935,91.024,434.692,174.402,21.547,153.626
C00647=1081.929,90.774,434.710,174.401,21.545,153.626
C00648=1081.924,90.525,434.728,174.399,21.542,153.626
C00649=1081.918,90.276,434.747,174.397,21.540,153.626
C00650=1081.913,90.027,434.765,174.395,21.538,153.626
C00651=1081.907,89.778,434.782,174.394,21.536,153.626
C00652=1081.901,89.528,434.800,174.391,21.534,153.625
C00653=1081.895,89.279,434.818,174.390,21.532,153.625
C00654=1081.889,89.029,434.836,174.388,21.529,153.625
C00655=1081.884,88.780,434.853,174.386,21.527,153.625
C00656=1081.878,88.531,434.871,174.385,21.526,153.625
C00657=1081.872,88.281,434.889,174.383,21.523,153.625
C00658=1081.867,88.032,434.906,174.382,21.521,153.625
C00659=1081.860,87.782,434.924,174.379,21.519,153.624
C00660=1081.855,87.533,434.942,174.378,21.517,153.624
C00661=1081.849,87.284,434.959,174.376,21.515,153.624
C00662=1081.843,87.035,434.977,174.374,21.513,153.624
C00663=1081.838,86.786,434.995,174.372,21.510,153.624
C00664=1081.832,86.536,435.013,174.371,21.508,153.624
C00665=1081.826,86.287,435.030,174.370,21.506,153.623
C00666=1081.821,86.038,435.048,174.367,21.503,153.623
C00667=1081.815,85.788,435.066,174.366,21.502,153.623
C00668=1081.809,85.539,435.083,174.364,21.499,153.623
C00669=1081.803,85.290,435.101,174.363,21.497,153.623
C00670=1081.797,85.040,435.119,174.360,21.495,153.623
C00671=1081.792,84.791,435.136,174.359,21.493,153.622
C00672=1081.786,84.542,435.154,174.357,21.491,153.622
C00673=1081.780,84.292,435.172,174.355,21.489,153.622
C00674=1081.775,84.043,435.189,174.354,21.487,153.622
C00675=1081.769,83.794,435.207,174.352,21.484,153.622
C00676=1081.764,83.545,435.224,174.351,21.482,153.621
C00677=1081.758,83.295,435.242,174.348,21.479,153.621
C00678=1081.752,83.046,435.259,174.347,21.477,153.621
C00679=1081.747,82.797,435.277,174.345,21.475,153.621
C00680=1081.741,82.547,435.295,174.344,21.473,153.621
C00681=1081.735,82.298,435.312,174.341,21.471,153.621
C00682=1081.730,82.049,435.330,174.340,21.468,153.620
C00683=1081.724,81.799,435.347,174.339,21.466,153.620
C00684=1081.718,81.550,435.365,174.337,21.464,153.620
C00685=1081.713,81.300,435.382,174.335,21.462,153.620
C00686=1081.707,81.051,435.400,174.333,21.460,153.620
C00687=1081.702,80.802,435.418,174.332,21.458,153.620
C00688=1081.696,80.552,435.435,174.330,21.455,153.619
C00689=1081.690,80.303,435.452,174.328,21.453,153.619
C00690=1081.684,80.054,435.469,174.327,21.451,153.619
C00691=1081.679,79.805,435.487,174.325,21.449,153.619
C00692=1081.673,79.525,435.507,174.323,21.446,153.619
C00693=1081.666,79.246,435.526,174.321,21.444,153.618
C00694=1081.660,78.966,435.545,174.319,21.441,153.618
C00695=1081.653,78.687,435.565,174.317,21.438,153.618
C00696=1081.648,78.437,435.582,174.316,21.437,153.618
C00697=1081.642,78.187,435.600,174.314,21.434,153.618
C00698=1081.636,77.938,435.618,174.312,21.432,153.617
C00699=1081.630,77.689,435.634,174.311,21.430,153.617
C00700=1081.625,77.440,435.651,174.309,21.427,153.617
C00701=1081.619,77.190,435.669,174.308,21.425,153.617
C00702=1081.614,76.941,435.686,174.305,21.423,153.617
C00703=1081.607,76.692,435.703,174.304,21.421,153.617
C00704=1081.602,76.443,435.721,174.303,21.419,153.616
C00705=1081.597,76.193,435.738,174.301,21.416,153.616
C00706=1081.590,75.944,435.755,174.299,21.414,153.616
C00707=1081.584,75.695,435.772,174.297,21.412,153.616
C00708=1081.579,75.445,435.789,174.296,21.410,153.616
C00709=1081.574,75.196,435.807,174.294,21.408,153.615
C00710=1081.567,74.946,435.823,174.292,21.406,153.615
C00711=1081.561,74.697,435.841,174.291,21.403,153.615
C00712=1081.556,74.448,435.859,174.289,21.401,153.615
C00713=1081.550,74.198,435.875,174.287,21.399,153.615
C00714=1081.544,73.949,435.892,174.285,21.396,153.615
C00715=1081.539,73.700,435.909,174.284,21.395,153.614
C00716=1081.533,73.450,435.927,174.283,21.392,153.614
C00717=1081.527,73.201,435.943,174.281,21.390,153.614
C00718=1081.522,72.952,435.961,174.279,21.388,153.614
C00719=1081.516,72.702,435.978,174.277,21.385,153.614
C00720=1081.510,72.453,435.995,174.276,21.383,153.613
C00721=1081.505,72.204,436.012,174.275,21.381,153.613
C00722=1081.499,71.954,436.030,174.272,21.379,153.613
C00723=1081.493,71.704,436.046,174.271,21.377,153.613
C00724=1081.487,71.455,436.063,174.269,21.374,153.613
C00725=1081.482,71.206,436.080,174.268,21.372,153.612
C00726=1081.476,70.957,436.097,174.266,21.370,153.612
C00727=1081.471,70.707,436.114,174.264,21.367,153.612
C00728=1081.464,70.459,436.131,174.263,21.365,153.612
C00729=1081.459,70.208,436.148,174.261,21.363,153.612
C00730=1081.453,69.959,436.166,174.259,21.361,153.612
C00731=1081.447,69.710,436.182,174.258,21.359,153.611
C00732=1081.442,69.460,436.199,174.256,21.356,153.611
C00733=1081.436,69.212,436.216,174.255,21.354,153.611
C00734=1081.430,68.962,436.233,174.253,21.352,153.611
C00735=1081.424,68.713,436.250,174.251,21.349,153.611
C00736=1081.419,68.463,436.267,174.250,21.348,153.610
C00737=1081.414,68.214,436.283,174.248,21.345,153.610
C00738=1081.407,67.964,436.301,174.246,21.343,153.610
C00739=1081.402,67.715,436.318,174.245,21.341,153.610
C00740=1081.396,67.465,436.334,174.243,21.338,153.610
C00741=1081.390,67.216,436.352,174.242,21.336,153.610
C00742=1081.384,66.967,436.368,174.240,21.333,153.609
C00743=1081.379,66.717,436.385,174.238,21.332,153.609
C00744=1081.373,66.469,436.402,174.237,21.330,153.609
C00745=1081.368,66.219,436.418,174.235,21.327,153.609
C00746=1081.362,65.970,436.435,174.234,21.325,153.608
C00747=1081.355,65.721,436.452,174.232,21.323,153.608
C00748=1081.350,65.471,436.469,174.230,21.320,153.608
C00749=1081.344,65.221,436.485,174.229,21.318,153.608
C00750=1081.338,64.971,436.502,174.227,21.316,153.608
C00751=1081.332,64.723,436.519,174.225,21.314,153.608
C00752=1081.327,64.473,436.536,174.224,21.312,153.607
C00753=1081.321,64.224,436.552,174.222,21.309,153.607
C00754=1081.315,63.974,436.568,174.221,21.307,153.607
C00755=1081.310,63.725,436.585,174.219,21.305,153.607
C00756=1081.303,63.445,436.604,174.217,21.302,153.607
C00757=1081.296,63.165,436.623,174.215,21.300,153.606
C00758=1081.290,62.887,436.641,174.214,21.298,153.606
C00759=1081.283,62.607,436.660,174.212,21.295,153.606
C00760=1081.278,62.357,436.676,174.210,21.293,153.606
C00761=1081.272,62.108,436.692,174.208,21.290,153.606
C00762=1081.265,61.859,436.709,174.207,21.288,153.605
C00763=1081.260,61.609,436.727,174.205,21.286,153.605
C00764=1081.254,61.360,436.743,174.203,21.283,153.605
C00765=1081.248,61.110,436.759,174.202,21.282,153.605
C00766=1081.242,60.861,436.775,174.200,21.279,153.605
C00767=1081.236,60.611,436.792,174.199,21.277,153.605
C00768=1081.231,60.362,436.809,174.197,21.275,153.604
C00769=1081.225,60.112,436.825,174.195,21.272,153.604
C00770=1081.218,59.864,436.842,174.194,21.270,153.604
C00771=1081.213,59.614,436.859,174.193,21.268,153.604
C00772=1081.207,59.365,436.875,174.191,21.266,153.603
C00773=1081.201,59.115,436.891,174.189,21.264,153.603
C00774=1081.195,58.866,436.907,174.187,21.261,153.603
C00775=1081.189,58.617,436.924,174.186,21.259,153.603
C00776=1081.184,58.367,436.940,174.185,21.257,153.603
C00777=1081.178,58.118,436.957,174.182,21.254,153.603
C00778=1081.172,57.868,436.973,174.181,21.252,153.602
C00779=1081.166,57.619,436.989,174.180,21.250,153.602
C00780=1081.161,57.369,437.006,174.178,21.248,153.602
C00781=1081.155,57.120,437.022,174.176,21.246,153.602
C00782=1081.149,56.871,437.039,174.175,21.244,153.602
C00783=1081.143,56.621,437.055,174.173,21.241,153.601
C00784=1081.137,56.372,437.071,174.172,21.239,153.601
C00785=1081.131,56.123,437.087,174.170,21.237,153.601
C00786=1081.126,55.873,437.104,174.168,21.234,153.601
C00787=1081.120,55.624,437.120,174.167,21.232,153.601
C00788=1081.114,55.374,437.137,174.165,21.230,153.600
C00789=1081.108,55.125,437.153,174.163,21.228,153.600
C00790=1081.102,54.876,437.169,174.162,21.225,153.600
C00791=1081.096,54.626,437.185,174.160,21.223,153.600
C00792=1081.092,54.377,437.201,174.159,21.221,153.600
C00793=1081.086,54.127,437.218,174.158,21.218,153.599
C00794=1081.080,53.878,437.234,174.155,21.216,153.599
C00795=1081.074,53.629,437.250,174.154,21.214,153.599
C00796=1081.068,53.379,437.266,174.153,21.211,153.599
C00797=1081.062,53.130,437.283,174.151,21.209,153.599
C00798=1081.057,52.880,437.299,174.149,21.207,153.598
C00799=1081.051,52.631,437.316,174.148,21.205,153.598
C00800=1081.045,52.381,437.331,174.146,21.202,153.598
C00801=1081.039,52.132,437.347,174.145,21.200,153.598
C00802=1081.034,51.882,437.364,174.144,21.198,153.597
C00803=1081.028,51.634,437.380,174.141,21.195,153.597
C00804=1081.022,51.384,437.396,174.140,21.193,153.597
C00805=1081.016,51.135,437.412,174.139,21.191,153.597
C00806=1081.011,50.885,437.428,174.137,21.189,153.597
C00807=1081.005,50.635,437.445,174.136,21.187,153.597
C00808=1080.999,50.386,437.461,174.134,21.184,153.596
C00809=1080.993,50.137,437.477,174.132,21.182,153.596
C00810=1080.988,49.888,437.493,174.131,21.179,153.596
C00811=1080.983,49.638,437.508,174.130,21.177,153.596
C00812=1080.977,49.389,437.525,174.128,21.175,153.596
C00813=1080.971,49.139,437.541,174.126,21.172,153.595
C00814=1080.965,48.889,437.557,174.125,21.170,153.595
C00815=1080.959,48.640,437.573,174.123,21.168,153.595
C00816=1080.954,48.391,437.589,174.122,21.166,153.595
C00817=1080.948,48.142,437.605,174.120,21.164,153.594
C00818=1080.943,47.892,437.621,174.118,21.161,153.594
C00819=1080.937,47.642,437.637,174.117,21.159,153.594
C00820=1080.931,47.363,437.655,174.115,21.156,153.594
C00821=1080.924,47.083,437.672,174.114,21.153,153.593
C00822=1080.918,46.803,437.691,174.112,21.151,153.593
C00823=1080.911,46.523,437.709,174.111,21.148,153.593
C00824=1080.906,46.273,437.724,174.108,21.146,153.593
C00825=1080.900,46.024,437.741,174.107,21.144,153.593
C00826=1080.894,45.775,437.757,174.106,21.142,153.592
C00827=1080.889,45.525,437.772,174.104,21.139,153.592
C00828=1080.883,45.276,437.788,174.103,21.137,153.592
C00829=1080.877,45.027,437.805,174.102,21.134,153.592
C00830=1080.872,44.777,437.820,174.099,21.132,153.592
C00831=1080.866,44.528,437.836,174.098,21.130,153.591
C00832=1080.861,44.278,437.852,174.097,21.127,153.591
C00833=1080.855,44.028,437.868,174.095,21.125,153.591
C00834=1080.850,43.779,437.884,174.094,21.123,153.591
C00835=1080.843,43.530,437.899,174.092,21.121,153.590
C00836=1080.837,43.281,437.916,174.090,21.118,153.590
C00837=1080.832,43.031,437.931,174.089,21.116,153.590
C00838=1080.826,42.782,437.947,174.088,21.114,153.590
C00839=1080.821,42.532,437.963,174.086,21.111,153.590
C00840=1080.815,42.283,437.979,174.084,21.109,153.589
C00841=1080.809,42.033,437.994,174.083,21.107,153.589
C00842=1080.802,41.784,438.010,174.081,21.104,153.589
C00843=1080.797,41.535,438.025,174.080,21.102,153.589
C00844=1080.791,41.285,438.041,174.078,21.100,153.589
C00845=1080.786,41.035,438.057,174.076,21.097,153.588
C00846=1080.780,40.786,438.073,174.075,21.095,153.588
C00847=1080.775,40.537,438.088,174.074,21.093,153.588
C00848=1080.768,40.288,438.104,174.073,21.091,153.588
C00849=1080.762,40.038,438.120,174.070,21.088,153.588
C00850=1080.757,39.788,438.135,174.069,21.086,153.587
C00851=1080.751,39.539,438.151,174.068,21.084,153.587
C00852=1080.746,39.289,438.167,174.066,21.081,153.587
C00853=1080.740,39.040,438.183,174.065,21.079,153.587
C00854=1080.734,38.791,438.197,174.063,21.077,153.586
C00855=1080.728,38.541,438.214,174.061,21.074,153.586
C00856=1080.722,38.291,438.229,174.060,21.072,153.586
C00857=1080.717,38.042,438.244,174.059,21.070,153.586
C00858=1080.711,37.793,438.260,174.057,21.067,153.586
C00859=1080.705,37.543,438.276,174.055,21.065,153.585
C00860=1080.699,37.293,438.291,174.054,21.063,153.585
C00861=1080.693,37.045,438.306,174.053,21.061,153.585
C00862=1080.688,36.795,438.322,174.051,21.058,153.585
C00863=1080.682,36.545,438.338,174.050,21.056,153.585
C00864=1080.676,36.297,438.353,174.048,21.054,153.584
C00865=1080.670,36.047,438.368,174.046,21.051,153.584
C00866=1080.665,35.797,438.384,174.045,21.049,153.584
C00867=1080.658,35.548,438.400,174.044,21.047,153.584
C00868=1080.653,35.298,438.415,174.042,21.044,153.583
C00869=1080.647,35.048,438.430,174.040,21.042,153.583
C00870=1080.641,34.799,438.446,174.039,21.040,153.583
C00871=1080.635,34.550,438.461,174.038,21.038,153.583
C00872=1080.629,34.300,438.476,174.036,21.035,153.583
C00873=1080.623,34.050,438.492,174.034,21.033,153.583
C00874=1080.618,33.802,438.507,174.033,21.031,153.582
C00875=1080.612,33.552,438.522,174.031,21.028,153.582
C00876=1080.606,33.302,438.538,174.030,21.026,153.582
C00877=1080.601,33.053,438.553,174.029,21.024,153.582
C00878=1080.594,32.804,438.569,174.027,21.022,153.581
C00879=1080.589,32.554,438.584,174.025,21.019,153.581
C00880=1080.583,32.305,438.599,174.024,21.017,153.581
C00881=1080.577,32.055,438.614,174.023,21.015,153.581
C00882=1080.572,31.806,438.630,174.021,21.012,153.581
C00883=1080.566,31.557,438.645,174.019,21.010,153.580
C00884=1080.560,31.277,438.662,174.018,21.008,153.580
C00885=1080.553,30.996,438.680,174.016,21.005,153.580
C00886=1080.546,30.717,438.697,174.014,21.002,153.580
C00887=1080.540,30.437,438.713,174.013,21.000,153.579
C00888=1080.534,30.187,438.729,174.012,20.997,153.579
C00889=1080.528,29.938,438.744,174.010,20.995,153.579
C00890=1080.523,29.689,438.760,174.008,20.993,153.579
C00891=1080.516,29.439,438.775,174.007,20.991,153.578
C00892=1080.511,29.190,438.790,174.005,20.988,153.578
C00893=1080.505,28.940,438.805,174.004,20.986,153.578
C00894=1080.499,28.690,438.820,174.003,20.984,153.578
C00895=1080.493,28.441,438.835,174.001,20.982,153.578
C00896=1080.488,28.191,438.850,173.999,20.979,153.577
C00897=1080.482,27.943,438.865,173.998,20.977,153.577
C00898=1080.476,27.693,438.880,173.997,20.975,153.577
C00899=1080.470,27.443,438.895,173.995,20.972,153.577
C00900=1080.465,27.194,438.911,173.993,20.970,153.577
C00901=1080.459,26.944,438.926,173.992,20.967,153.576
C00902=1080.453,26.695,438.941,173.991,20.966,153.576
C00903=1080.447,26.445,438.956,173.989,20.963,153.576
C00904=1080.441,26.195,438.971,173.988,20.961,153.576
C00905=1080.436,25.946,438.986,173.986,20.959,153.576
C00906=1080.429,25.696,439.001,173.985,20.957,153.575
C00907=1080.423,25.447,439.015,173.983,20.954,153.575
C00908=1080.418,25.198,439.031,173.982,20.952,153.575
C00909=1080.412,24.949,439.045,173.981,20.949,153.575
C00910=1080.406,24.699,439.061,173.978,20.947,153.575
C00911=1080.401,24.450,439.076,173.977,20.945,153.574
C00912=1080.394,24.200,439.090,173.976,20.942,153.574
C00913=1080.389,23.950,439.106,173.975,20.940,153.574
C00914=1080.383,23.701,439.121,173.973,20.938,153.574
C00915=1080.376,23.451,439.136,173.971,20.936,153.573
C00916=1080.371,23.202,439.151,173.970,20.934,153.573
C00917=1080.365,22.952,439.166,173.969,20.931,153.573
C00918=1080.359,22.704,439.180,173.967,20.929,153.573
C00919=1080.354,22.454,439.196,173.966,20.927,153.573
C00920=1080.348,22.205,439.210,173.964,20.924,153.572
C00921=1080.341,21.955,439.225,173.963,20.922,153.572
C00922=1080.337,21.705,439.240,173.961,20.920,153.572
C00923=1080.330,21.455,439.255,173.960,20.917,153.572
C00924=1080.325,21.206,439.269,173.958,20.915,153.572
C00925=1080.319,20.956,439.285,173.957,20.913,153.571
C00926=1080.313,20.708,439.299,173.955,20.910,153.571
C00927=1080.307,20.458,439.314,173.954,20.908,153.571
C00928=1080.302,20.208,439.329,173.953,20.906,153.571
C00929=1080.296,19.958,439.344,173.951,20.904,153.571
C00930=1080.290,19.709,439.358,173.950,20.901,153.570
C00931=1080.283,19.460,439.373,173.948,20.899,153.570
C00932=1080.278,19.210,439.388,173.947,20.897,153.570
C00933=1080.272,18.960,439.403,173.945,20.894,153.570
C00934=1080.267,18.711,439.417,173.944,20.892,153.569
C00935=1080.260,18.462,439.432,173.942,20.890,153.569
C00936=1080.255,18.212,439.447,173.941,20.888,153.569
C00937=1080.249,17.963,439.462,173.939,20.885,153.569
C00938=1080.243,17.713,439.476,173.938,20.883,153.569
C00939=1080.237,17.463,439.491,173.937,20.881,153.568
C00940=1080.231,17.214,439.506,173.935,20.879,153.568
C00941=1080.226,16.965,439.521,173.933,20.876,153.568
C00942=1080.220,16.715,439.535,173.932,20.874,153.568
C00943=1080.214,16.466,439.550,173.931,20.872,153.568
C00944=1080.208,16.216,439.565,173.930,20.869,153.567
C00945=1080.202,15.967,439.579,173.927,20.867,153.567
C00946=1080.196,15.717,439.593,173.926,20.865,153.567
C00947=1080.191,15.468,439.609,173.925,20.863,153.567
C00948=1080.184,15.190,439.625,173.923,20.860,153.566
C00949=1080.177,14.911,439.641,173.922,20.858,153.566
C00950=1080.171,14.632,439.657,173.920,20.855,153.566
C00951=1080.165,14.354,439.673,173.918,20.853,153.566
C00952=1080.159,14.104,439.688,173.917,20.850,153.566
C00953=1080.153,13.855,439.703,173.915,20.848,153.565
C00954=1080.147,13.605,439.717,173.914,20.846,153.565
C00955=1080.141,13.356,439.731,173.913,20.843,153.565
C00956=1080.135,13.107,439.746,173.911,20.841,153.565
C00957=1080.129,12.857,439.760,173.909,20.839,153.565
C00958=1080.123,12.608,439.775,173.908,20.836,153.564
C00959=1080.117,12.357,439.789,173.907,20.834,153.564
C00960=1080.112,12.109,439.804,173.905,20.832,153.564
C00961=1080.105,11.858,439.818,173.903,20.830,153.564
C00962=1080.100,11.609,439.832,173.902,20.828,153.564
C00963=1080.093,11.360,439.847,173.901,20.826,153.563
C00964=1080.088,11.110,439.861,173.900,20.824,153.563
C00965=1080.082,10.861,439.876,173.898,20.821,153.563
C00966=1080.076,10.611,439.890,173.896,20.819,153.563
C00967=1080.070,10.362,439.905,173.895,20.817,153.563
C00968=1080.064,10.112,439.919,173.894,20.814,153.562
C00969=1080.058,9.863,439.933,173.893,20.812,153.562
C00970=1080.053,9.613,439.947,173.890,20.810,153.562
C00971=1080.046,9.364,439.962,173.889,20.807,153.562
C00972=1080.040,9.114,439.976,173.888,20.805,153.562
C00973=1080.034,8.865,439.990,173.887,20.803,153.561
C00974=1080.028,8.615,440.004,173.885,20.801,153.561
C00975=1080.023,8.366,440.019,173.883,20.798,153.561
C00976=1080.017,8.116,440.033,173.882,20.796,153.561
C00977=1080.011,7.867,440.048,173.881,20.794,153.561
C00978=1080.005,7.617,440.062,173.879,20.792,153.560
C00979=1079.999,7.367,440.076,173.878,20.790,153.560
C00980=1079.993,7.118,440.090,173.876,20.788,153.560
C00981=1079.988,6.868,440.104,173.875,20.785,153.560
C00982=1079.982,6.619,440.119,173.873,20.783,153.560
C00983=1079.976,6.369,440.133,173.872,20.781,153.559
C00984=1079.971,6.120,440.147,173.871,20.778,153.559
C00985=1079.964,5.870,440.161,173.869,20.776,153.559
C00986=1079.958,5.621,440.175,173.868,20.774,153.559
C00987=1079.952,5.372,440.190,173.866,20.771,153.559
C00988=1079.946,5.121,440.204,173.865,20.769,153.558
C00989=1079.941,4.872,440.218,173.863,20.767,153.558
C00990=1079.935,4.623,440.232,173.862,20.765,153.558
C00991=1079.929,4.373,440.246,173.860,20.762,153.558
C00992=1079.923,4.123,440.261,173.859,20.760,153.558
C00993=1079.918,3.874,440.275,173.858,20.758,153.557
C00994=1079.911,3.625,440.288,173.856,20.756,153.557
C00995=1079.905,3.374,440.303,173.855,20.754,153.557
C00996=1079.899,3.126,440.317,173.853,20.751,153.557
C00997=1079.894,2.876,440.331,173.852,20.749,153.557
C00998=1079.889,2.626,440.345,173.850,20.747,153.556
C00999=1079.882,2.376,440.359,173.849,20.745,153.556
C01000=1079.877,2.127,440.374,173.847,20.742,153.556
C01001=1079.871,1.878,440.388,173.846,20.740,153.556
C01002=1079.865,1.628,440.401,173.845,20.738,153.555
C01003=1079.859,1.378,440.415,173.844,20.736,153.555
C01004=1079.853,1.129,440.430,173.842,20.734,153.555
C01005=1079.848,0.880,440.444,173.840,20.731,153.555
C01006=1079.842,0.630,440.457,173.839,20.729,153.555
C01007=1079.837,0.380,440.471,173.838,20.727,153.555
C01008=1079.830,0.131,440.486,173.837,20.724,153.554
C01009=1079.824,-0.119,440.499,173.834,20.722,153.554
C01010=1079.819,-0.368,440.513,173.833,20.720,153.554
C01011=1079.813,-0.618,440.527,173.832,20.717,153.554
C01012=1079.806,-0.894,440.543,173.831,20.715,153.553
C01013=1079.800,-1.171,440.558,173.829,20.712,153.553
C01014=1079.794,-1.447,440.574,173.827,20.710,153.553
C01015=1079.788,-1.724,440.589,173.825,20.707,153.553
C01016=1079.782,-1.974,440.603,173.824,20.705,153.553
C01017=1079.776,-2.223,440.618,173.823,20.703,153.552
C01018=1079.770,-2.472,440.631,173.822,20.701,153.552
C01019=1079.764,-2.722,440.645,173.820,20.699,153.552
C01020=1079.759,-2.971,440.659,173.818,20.696,153.552
C01021=1079.753,-3.221,440.673,173.817,20.694,153.552
C01022=1079.746,-3.471,440.686,173.816,20.692,153.551
C01023=1079.741,-3.720,440.700,173.814,20.689,153.551
C01024=1079.735,-3.970,440.714,173.813,20.687,153.551
C01025=1079.729,-4.219,440.727,173.811,20.685,153.551
C01026=1079.723,-4.468,440.742,173.810,20.683,153.551
C01027=1079.717,-4.718,440.755,173.809,20.681,153.550
C01028=1079.711,-4.968,440.769,173.807,20.678,153.550
C01029=1079.705,-5.217,440.782,173.805,20.676,153.550
C01030=1079.699,-5.467,440.796,173.804,20.674,153.550
C01031=1079.693,-5.717,440.811,173.803,20.672,153.550
C01032=1079.687,-5.966,440.824,173.802,20.670,153.549
C01033=1079.682,-6.216,440.838,173.800,20.667,153.549
C01034=1079.675,-6.465,440.851,173.798,20.665,153.549
C01035=1079.670,-6.715,440.865,173.797,20.663,153.549
C01036=1079.664,-6.964,440.878,173.796,20.661,153.549
C01037=1079.658,-7.214,440.892,173.795,20.659,153.548
C01038=1079.652,-7.464,440.906,173.792,20.656,153.548
C01039=1079.646,-7.713,440.919,173.791,20.654,153.548
C01040=1079.641,-7.962,440.933,173.790,20.653,153.548
C01041=1079.634,-8.212,440.947,173.789,20.650,153.548
C01042=1079.629,-8.461,440.960,173.787,20.648,153.547
C01043=1079.622,-8.711,440.974,173.785,20.646,153.547
C01044=1079.617,-8.961,440.988,173.784,20.644,153.547
C01045=1079.610,-9.210,441.001,173.783,20.642,153.547
C01046=1079.605,-9.460,441.014,173.782,20.639,153.547
C01047=1079.599,-9.710,441.028,173.780,20.637,153.547
C01048=1079.593,-9.959,441.042,173.778,20.635,153.546
C01049=1079.587,-10.208,441.055,173.777,20.633,153.546
C01050=1079.582,-10.458,441.069,173.776,20.630,153.546
C01051=1079.575,-10.708,441.082,173.774,20.628,153.546
C01052=1079.569,-10.958,441.096,173.773,20.626,153.546
C01053=1079.563,-11.207,441.109,173.771,20.624,153.545
C01054=1079.558,-11.456,441.123,173.770,20.622,153.545
C01055=1079.552,-11.706,441.136,173.769,20.619,153.545
C01056=1079.546,-11.956,441.150,173.767,20.617,153.545
C01057=1079.540,-12.205,441.163,173.766,20.615,153.545
C01058=1079.535,-12.455,441.177,173.764,20.613,153.545
C01059=1079.528,-12.704,441.190,173.763,20.610,153.544
C01060=1079.523,-12.953,441.204,173.761,20.608,153.544
C01061=1079.517,-13.203,441.217,173.760,20.606,153.544
C01062=1079.512,-13.453,441.230,173.759,20.604,153.544
C01063=1079.505,-13.703,441.244,173.757,20.602,153.544
C01064=1079.499,-13.953,441.258,173.756,20.599,153.543
C01065=1079.493,-14.202,441.271,173.754,20.598,153.543
C01066=1079.488,-14.452,441.284,173.753,20.596,153.543
C01067=1079.482,-14.701,441.298,173.752,20.594,153.543
C01068=1079.476,-14.950,441.311,173.750,20.591,153.543
C01069=1079.470,-15.200,441.325,173.748,20.589,153.542
C01070=1079.464,-15.450,441.337,173.747,20.587,153.542
C01071=1079.458,-15.699,441.351,173.746,20.585,153.542
C01072=1079.452,-15.949,441.364,173.745,20.583,153.542
C01073=1079.446,-16.198,441.378,173.743,20.581,153.542
C01074=1079.440,-16.448,441.390,173.741,20.578,153.542
C01075=1079.435,-16.698,441.404,173.740,20.576,153.541
C01076=1079.428,-16.972,441.418,173.739,20.574,153.541
C01077=1079.421,-17.247,441.433,173.737,20.571,153.541
C01078=1079.414,-17.522,441.447,173.735,20.569,153.541
C01079=1079.408,-17.797,441.462,173.734,20.567,153.541
C01080=1079.402,-18.046,441.476,173.732,20.564,153.540
C01081=1079.397,-18.296,441.489,173.731,20.562,153.540
C01082=1079.390,-18.546,441.502,173.729,20.560,153.540
C01083=1079.384,-18.795,441.515,173.728,20.558,153.540
C01084=1079.378,-19.045,441.528,173.727,20.556,153.540
C01085=1079.373,-19.294,441.542,173.726,20.554,153.540
C01086=1079.367,-19.544,441.554,173.723,20.552,153.539
C01087=1079.361,-19.794,441.568,173.722,20.549,153.539
C01088=1079.355,-20.043,441.581,173.721,20.547,153.539
C01089=1079.349,-20.293,441.594,173.720,20.545,153.539
C01090=1079.343,-20.542,441.607,173.718,20.543,153.539
C01091=1079.337,-20.792,441.620,173.716,20.541,153.539
C01092=1079.331,-21.041,441.633,173.715,20.539,153.538
C01093=1079.326,-21.291,441.647,173.714,20.537,153.538
C01094=1079.320,-21.541,441.659,173.712,20.535,153.538
C01095=1079.313,-21.790,441.673,173.711,20.533,153.538
C01096=1079.308,-22.040,441.685,173.710,20.531,153.538
C01097=1079.301,-22.289,441.699,173.708,20.528,153.537
C01098=1079.296,-22.540,441.712,173.706,20.526,153.537
C01099=1079.290,-22.789,441.725,173.705,20.524,153.537
C01100=1079.284,-23.039,441.738,173.704,20.522,153.537
C01101=1079.278,-23.288,441.751,173.703,20.520,153.537
C01102=1079.272,-23.538,441.763,173.701,20.518,153.537
C01103=1079.266,-23.787,441.777,173.699,20.516,153.536
C01104=1079.261,-24.037,441.789,173.698,20.514,153.536
C01105=1079.255,-24.286,441.803,173.697,20.512,153.536
C01106=1079.249,-24.536,441.815,173.695,20.509,153.536
C01107=1079.243,-24.785,441.829,173.694,20.507,153.536
C01108=1079.238,-25.035,441.842,173.693,20.505,153.535
C01109=1079.231,-25.284,441.855,173.691,20.503,153.535
C01110=1079.225,-25.534,441.867,173.689,20.501,153.535
C01111=1079.219,-25.784,441.881,173.688,20.499,153.535
C01112=1079.213,-26.033,441.893,173.687,20.497,153.535
C01113=1079.207,-26.283,441.907,173.686,20.495,153.535
C01114=1079.202,-26.533,441.920,173.684,20.493,153.535
C01115=1079.197,-26.782,441.932,173.682,20.490,153.534
C01116=1079.190,-27.031,441.945,173.681,20.488,153.534
C01117=1079.185,-27.281,441.958,173.680,20.486,153.534
C01118=1079.178,-27.531,441.971,173.678,20.484,153.534
C01119=1079.172,-27.780,441.984,173.677,20.482,153.534
C01120=1079.166,-28.030,441.996,173.676,20.481,153.534
C01121=1079.160,-28.280,442.009,173.673,20.478,153.533
C01122=1079.154,-28.529,442.022,173.672,20.476,153.533
C01123=1079.148,-28.779,442.034,173.671,20.474,153.533
C01124=1079.142,-29.029,442.048,173.670,20.472,153.533
C01125=1079.136,-29.278,442.060,173.668,20.470,153.533
C01126=1079.130,-29.528,442.073,173.667,20.468,153.533
C01127=1079.124,-29.778,442.086,173.665,20.466,153.533
C01128=1079.118,-30.028,442.099,173.664,20.464,153.532
C01129=1079.113,-30.277,442.111,173.662,20.462,153.532
C01130=1079.107,-30.526,442.124,173.661,20.460,153.532
C01131=1079.101,-30.776,442.137,173.660,20.458,153.532
C01132=1079.095,-31.026,442.149,173.658,20.456,153.532
C01133=1079.089,-31.275,442.163,173.657,20.454,153.532
C01134=1079.082,-31.525,442.174,173.655,20.451,153.531
C01135=1079.076,-31.774,442.187,173.654,20.449,153.531
C01136=1079.070,-32.024,442.200,173.652,20.447,153.531
C01137=1079.065,-32.273,442.213,173.651,20.445,153.531
C01138=1079.059,-32.523,442.225,173.650,20.443,153.531
C01139=1079.053,-32.773,442.238,173.648,20.441,153.531
C01140=1079.046,-33.047,442.252,173.646,20.439,153.530
C01141=1079.040,-33.321,442.265,173.645,20.437,153.530
C01142=1079.033,-33.595,442.279,173.644,20.435,153.530
C01143=1079.027,-33.869,442.293,173.642,20.432,153.530
C01144=1079.021,-34.119,442.306,173.640,20.430,153.530
C01145=1079.015,-34.368,442.318,173.639,20.428,153.530
C01146=1079.009,-34.618,442.332,173.638,20.426,153.529
C01147=1079.004,-34.867,442.344,173.636,20.424,153.529
C01148=1078.998,-35.117,442.356,173.635,20.422,153.529
C01149=1078.991,-35.366,442.368,173.633,20.420,153.529
C01150=1078.985,-35.616,442.381,173.632,20.418,153.529
C01151=1078.979,-35.866,442.393,173.630,20.416,153.529
C01152=1078.974,-36.115,442.406,173.629,20.414,153.529
C01153=1078.968,-36.365,442.419,173.628,20.412,153.528
C01154=1078.962,-36.614,442.431,173.627,20.410,153.528
C01155=1078.956,-36.864,442.444,173.625,20.408,153.528
C01156=1078.951,-37.114,442.456,173.623,20.406,153.528
C01157=1078.945,-37.363,442.469,173.622,20.404,153.528
C01158=1078.939,-37.613,442.481,173.620,20.402,153.528
C01159=1078.932,-37.863,442.493,173.619,20.400,153.528
C01160=1078.926,-38.113,442.506,173.618,20.398,153.527
C01161=1078.921,-38.362,442.518,173.616,20.396,153.527
C01162=1078.915,-38.612,442.531,173.615,20.394,153.527
C01163=1078.909,-38.861,442.544,173.613,20.392,153.527
C01164=1078.902,-39.111,442.556,173.612,20.390,153.527
C01165=1078.897,-39.360,442.568,173.610,20.388,153.527
C01166=1078.891,-39.610,442.580,173.609,20.386,153.527
C01167=1078.885,-39.860,442.593,173.608,20.384,153.526
C01168=1078.878,-40.109,442.605,173.606,20.382,153.526
C01169=1078.873,-40.359,442.618,173.605,20.380,153.526
C01170=1078.867,-40.608,442.630,173.604,20.378,153.526
C01171=1078.861,-40.858,442.642,173.601,20.376,153.526
C01172=1078.855,-41.108,442.654,173.600,20.374,153.526
C01173=1078.849,-41.358,442.667,173.599,20.372,153.526
C01174=1078.843,-41.606,442.678,173.598,20.370,153.525
C01175=1078.837,-41.856,442.691,173.596,20.368,153.525
C01176=1078.831,-42.106,442.704,173.595,20.367,153.525
C01177=1078.825,-42.356,442.716,173.593,20.365,153.525
C01178=1078.819,-42.605,442.728,173.592,20.363,153.525
C01179=1078.813,-42.855,442.740,173.590,20.361,153.525
C01180=1078.807,-43.105,442.753,173.589,20.359,153.525
C01181=1078.801,-43.355,442.764,173.587,20.357,153.525
C01182=1078.795,-43.604,442.776,173.586,20.355,153.524
C01183=1078.790,-43.854,442.789,173.585,20.353,153.524
C01184=1078.783,-44.104,442.801,173.583,20.351,153.524
C01185=1078.777,-44.353,442.813,173.582,20.350,153.524
C01186=1078.771,-44.602,442.825,173.581,20.348,153.524
C01187=1078.765,-44.852,442.837,173.578,20.345,153.524
C01188=1078.759,-45.102,442.850,173.577,20.343,153.524
C01189=1078.753,-45.351,442.862,173.576,20.341,153.523
C01190=1078.747,-45.601,442.874,173.574,20.340,153.523
C01191=1078.742,-45.851,442.886,173.573,20.338,153.523
C01192=1078.736,-46.100,442.898,173.572,20.336,153.523
C01193=1078.730,-46.350,442.910,173.570,20.334,153.523
C01194=1078.724,-46.600,442.923,173.569,20.332,153.523
C01195=1078.718,-46.849,442.934,173.568,20.330,153.523
C01196=1078.712,-47.099,442.947,173.566,20.328,153.523
C01197=1078.705,-47.349,442.958,173.564,20.326,153.522
C01198=1078.700,-47.598,442.970,173.563,20.324,153.522
C01199=1078.694,-47.848,442.983,173.561,20.322,153.522
C01200=1078.688,-48.098,442.995,173.560,20.320,153.522
C01201=1078.682,-48.347,443.007,173.559,20.318,153.522
C01202=1078.676,-48.597,443.018,173.557,20.317,153.522
C01203=1078.670,-48.847,443.031,173.556,20.315,153.522
C01204=1078.664,-49.121,443.044,173.554,20.312,153.522
C01205=1078.657,-49.395,443.057,173.553,20.310,153.521
C01206=1078.650,-49.670,443.070,173.551,20.308,153.521
C01207=1078.644,-49.944,443.084,173.549,20.306,153.521
C01208=1078.638,-50.193,443.095,173.548,20.304,153.521
C01209=1078.632,-50.443,443.108,173.546,20.303,153.521
C01210=1078.626,-50.693,443.119,173.545,20.301,153.521
C01211=1078.621,-50.943,443.131,173.544,20.299,153.521
C01212=1078.614,-51.192,443.143,173.542,20.297,153.521
C01213=1078.607,-51.442,443.155,173.541,20.295,153.520
C01214=1078.602,-51.691,443.167,173.540,20.294,153.520
C01215=1078.596,-51.941,443.179,173.538,20.292,153.520
C01216=1078.589,-52.191,443.190,173.537,20.290,153.520
C01217=1078.584,-52.440,443.202,173.535,20.288,153.520
C01218=1078.577,-52.690,443.214,173.533,20.286,153.520
C01219=1078.571,-52.940,443.226,173.532,20.284,153.520
C01220=1078.566,-53.189,443.237,173.530,20.283,153.520
C01221=1078.559,-53.439,443.249,173.529,20.281,153.520
C01222=1078.553,-53.689,443.261,173.528,20.279,153.520
C01223=1078.548,-53.938,443.273,173.526,20.277,153.520
C01224=1078.541,-54.188,443.285,173.525,20.275,153.519
C01225=1078.535,-54.438,443.296,173.523,20.274,153.519
C01226=1078.529,-54.687,443.308,173.522,20.272,153.519
C01227=1078.523,-54.937,443.320,173.521,20.270,153.519
C01228=1078.517,-55.186,443.331,173.519,20.268,153.519
C01229=1078.510,-55.436,443.343,173.517,20.266,153.519
C01230=1078.504,-55.686,443.355,173.516,20.264,153.519
C01231=1078.499,-55.935,443.366,173.514,20.263,153.519
C01232=1078.492,-56.185,443.378,173.513,20.261,153.519
C01233=1078.486,-56.435,443.390,173.512,20.259,153.519
C01234=1078.480,-56.684,443.402,173.510,20.258,153.518
C01235=1078.474,-56.934,443.413,173.509,20.256,153.518
C01236=1078.468,-57.183,443.425,173.507,20.254,153.518
C01237=1078.462,-57.434,443.436,173.506,20.252,153.518
C01238=1078.456,-57.683,443.448,173.505,20.251,153.518
C01239=1078.450,-57.933,443.459,173.503,20.249,153.518
C01240=1078.444,-58.183,443.472,173.501,20.247,153.518
C01241=1078.438,-58.432,443.483,173.500,20.245,153.518
C01242=1078.432,-58.682,443.495,173.498,20.243,153.518
C01243=1078.426,-58.931,443.506,173.497,20.241,153.518
C01244=1078.420,-59.181,443.518,173.495,20.240,153.518
C01245=1078.414,-59.431,443.529,173.494,20.238,153.517
C01246=1078.408,-59.680,443.541,173.493,20.236,153.517
C01247=1078.401,-59.930,443.552,173.491,20.234,153.517
C01248=1078.396,-60.180,443.564,173.490,20.233,153.517
C01249=1078.390,-60.430,443.576,173.488,20.231,153.517
C01250=1078.384,-60.679,443.587,173.487,20.229,153.517
C01251=1078.377,-60.929,443.598,173.485,20.228,153.517
C01252=1078.372,-61.178,443.611,173.484,20.226,153.517
C01253=1078.366,-61.428,443.622,173.483,20.224,153.517
C01254=1078.360,-61.678,443.633,173.481,20.222,153.517
C01255=1078.353,-61.927,443.645,173.479,20.221,153.517
C01256=1078.347,-62.177,443.656,173.478,20.219,153.516
C01257=1078.341,-62.427,443.668,173.476,20.217,153.516
C01258=1078.336,-62.676,443.679,173.475,20.215,153.516
C01259=1078.329,-62.926,443.690,173.473,20.214,153.516
C01260=1078.323,-63.175,443.702,173.472,20.212,153.516
C01261=1078.317,-63.425,443.713,173.471,20.210,153.516
C01262=1078.312,-63.675,443.725,173.469,20.209,153.516
C01263=1078.305,-63.925,443.736,173.468,20.207,153.516
C01264=1078.300,-64.174,443.747,173.466,20.205,153.516
C01265=1078.293,-64.424,443.759,173.465,20.203,153.516
C01266=1078.287,-64.673,443.770,173.464,20.202,153.516
C01267=1078.282,-64.923,443.782,173.462,20.200,153.516
C01268=1078.275,-65.199,443.794,173.460,20.198,153.516
C01269=1078.269,-65.475,443.807,173.459,20.196,153.515
C01270=1078.262,-65.751,443.820,173.457,20.194,153.515
C01271=1078.256,-66.026,443.831,173.456,20.192,153.515
C01272=1078.249,-66.275,443.843,173.454,20.190,153.515
C01273=1078.244,-66.525,443.855,173.452,20.188,153.515
C01274=1078.238,-66.775,443.866,173.451,20.187,153.515
C01275=1078.232,-67.025,443.877,173.449,20.185,153.515
C01276=1078.225,-67.274,443.889,173.448,20.183,153.515
C01277=1078.219,-67.524,443.900,173.446,20.182,153.515
C01278=1078.214,-67.773,443.911,173.445,20.180,153.515
C01279=1078.207,-68.023,443.922,173.444,20.179,153.515
C01280=1078.202,-68.273,443.934,173.442,20.177,153.515
C01281=1078.196,-68.523,443.945,173.441,20.175,153.514
C01282=1078.190,-68.772,443.956,173.439,20.174,153.514
C01283=1078.184,-69.022,443.967,173.438,20.172,153.514
C01284=1078.178,-69.272,443.978,173.437,20.170,153.514
C01285=1078.172,-69.521,443.990,173.435,20.169,153.514
C01286=1078.166,-69.770,444.001,173.434,20.167,153.514
C01287=1078.161,-70.021,444.013,173.432,20.165,153.514
C01288=1078.155,-70.270,444.024,173.431,20.164,153.514
C01289=1078.148,-70.521,444.035,173.430,20.162,153.514
C01290=1078.142,-70.769,444.046,173.428,20.160,153.514
C01291=1078.137,-71.019,444.057,173.427,20.159,153.514
C01292=1078.130,-71.269,444.069,173.425,20.157,153.514
C01293=1078.125,-71.519,444.079,173.424,20.155,153.514
C01294=1078.119,-71.768,444.090,173.421,20.153,153.514
C01295=1078.113,-72.019,444.102,173.420,20.151,153.513
C01296=1078.107,-72.268,444.113,173.419,20.150,153.513
C01297=1078.102,-72.518,444.124,173.417,20.148,153.513
C01298=1078.095,-72.767,444.136,173.416,20.146,153.513
C01299=1078.089,-73.017,444.147,173.414,20.145,153.513
C01300=1078.084,-73.266,444.158,173.413,20.144,153.513
C01301=1078.077,-73.516,444.169,173.412,20.142,153.513
C01302=1078.072,-73.766,444.180,173.410,20.140,153.513
C01303=1078.066,-74.015,444.191,173.409,20.139,153.513
C01304=1078.059,-74.265,444.202,173.407,20.137,153.513
C01305=1078.054,-74.515,444.213,173.406,20.136,153.513
C01306=1078.048,-74.764,444.224,173.404,20.134,153.513
C01307=1078.042,-75.015,444.235,173.403,20.132,153.513
C01308=1078.036,-75.264,444.246,173.401,20.131,153.513
C01309=1078.030,-75.514,444.257,173.400,20.129,153.513
C01310=1078.024,-75.764,444.268,173.398,20.128,153.513
C01311=1078.018,-76.013,444.279,173.397,20.126,153.512
C01312=1078.012,-76.263,444.289,173.396,20.124,153.512
C01313=1078.005,-76.513,444.300,173.394,20.123,153.512
C01314=1078.000,-76.762,444.311,173.393,20.121,153.512
C01315=1077.994,-77.012,444.322,173.391,20.120,153.512
C01316=1077.987,-77.262,444.333,173.390,20.118,153.512
C01317=1077.982,-77.511,444.344,173.388,20.117,153.512
C01318=1077.976,-77.761,444.355,173.387,20.115,153.512
C01319=1077.970,-78.011,444.366,173.385,20.113,153.512
C01320=1077.963,-78.260,444.377,173.384,20.112,153.512
C01321=1077.957,-78.510,444.387,173.382,20.111,153.512
C01322=1077.952,-78.759,444.398,173.381,20.109,153.512
C01323=1077.945,-79.009,444.410,173.379,20.108,153.512
C01324=1077.940,-79.259,444.420,173.378,20.106,153.512
C01325=1077.934,-79.508,444.431,173.376,20.105,153.512
C01326=1077.928,-79.759,444.443,173.375,20.103,153.512
C01327=1077.921,-80.008,444.453,173.373,20.101,153.512
C01328=1077.915,-80.257,444.464,173.372,20.100,153.512
C01329=1077.909,-80.507,444.475,173.370,20.098,153.512
C01330=1077.903,-80.757,444.484,173.369,20.097,153.512
C01331=1077.897,-81.007,444.495,173.367,20.095,153.512
C01332=1077.890,-81.285,444.508,173.366,20.094,153.512
C01333=1077.883,-81.563,444.520,173.364,20.092,153.512
C01334=1077.876,-81.840,444.531,173.362,20.090,153.512
C01335=1077.870,-82.118,444.543,173.361,20.089,153.512
C01336=1077.863,-82.368,444.554,173.359,20.087,153.512
C01337=1077.857,-82.618,444.564,173.358,20.086,153.512
C01338=1077.851,-82.867,444.575,173.356,20.085,153.512
C01339=1077.845,-83.117,444.586,173.355,20.083,153.512
C01340=1077.838,-83.366,444.597,173.353,20.082,153.512
C01341=1077.833,-83.617,444.607,173.352,20.080,153.512
C01342=1077.827,-83.866,444.618,173.350,20.079,153.512
C01343=1077.820,-84.116,444.629,173.349,20.077,153.511
C01344=1077.814,-84.365,444.639,173.347,20.076,153.511
C01345=1077.809,-84.615,444.650,173.346,20.074,153.511
C01346=1077.802,-84.865,444.660,173.344,20.073,153.511
C01347=1077.796,-85.115,444.671,173.342,20.072,153.512
C01348=1077.790,-85.364,444.682,173.341,20.070,153.512
C01349=1077.784,-85.614,444.692,173.339,20.069,153.511
C01350=1077.778,-85.864,444.702,173.338,20.067,153.511
C01351=1077.771,-86.114,444.713,173.336,20.066,153.511
C01352=1077.766,-86.363,444.724,173.335,20.065,153.511
C01353=1077.760,-86.613,444.735,173.333,20.063,153.511
C01354=1077.754,-86.862,444.744,173.332,20.062,153.511
C01355=1077.747,-87.113,444.756,173.330,20.060,153.511
C01356=1077.742,-87.362,444.767,173.329,20.059,153.511
C01357=1077.735,-87.612,444.776,173.327,20.057,153.511
C01358=1077.730,-87.861,444.787,173.326,20.056,153.511
C01359=1077.723,-88.110,444.797,173.324,20.055,153.511
C01360=1077.717,-88.361,444.809,173.323,20.053,153.511
C01361=1077.711,-88.611,444.819,173.321,20.052,153.511
C01362=1077.705,-88.860,444.829,173.320,20.050,153.511
C01363=1077.699,-89.109,444.840,173.318,20.049,153.511
C01364=1077.693,-89.359,444.849,173.317,20.047,153.511
C01365=1077.687,-89.609,444.861,173.315,20.046,153.511
C01366=1077.680,-89.859,444.871,173.313,20.045,153.511
C01367=1077.675,-90.109,444.881,173.313,20.044,153.511
C01368=1077.669,-90.358,444.892,173.311,20.043,153.511
C01369=1077.663,-90.608,444.902,173.310,20.041,153.511
C01370=1077.657,-90.858,444.912,173.308,20.040,153.511
C01371=1077.650,-91.107,444.923,173.307,20.038,153.511
C01372=1077.645,-91.358,444.933,173.305,20.037,153.511
C01373=1077.638,-91.607,444.944,173.304,20.036,153.511
C01374=1077.633,-91.857,444.954,173.302,20.034,153.511
C01375=1077.627,-92.106,444.965,173.301,20.033,153.511
C01376=1077.620,-92.355,444.975,173.299,20.031,153.511
C01377=1077.615,-92.606,444.985,173.297,20.030,153.511
C01378=1077.608,-92.855,444.996,173.296,20.029,153.511
C01379=1077.603,-93.106,445.006,173.294,20.027,153.511
C01380=1077.596,-93.355,445.016,173.293,20.026,153.511
C01381=1077.591,-93.605,445.026,173.291,20.025,153.511
C01382=1077.584,-93.854,445.037,173.290,20.024,153.511
C01383=1077.579,-94.104,445.047,173.288,20.022,153.511
C01384=1077.572,-94.353,445.057,173.287,20.021,153.511
C01385=1077.566,-94.603,445.068,173.285,20.019,153.511
C01386=1077.561,-94.853,445.078,173.284,20.018,153.511
C01387=1077.555,-95.102,445.088,173.282,20.017,153.511
C01388=1077.549,-95.353,445.099,173.280,20.015,153.511
C01389=1077.542,-95.602,445.109,173.279,20.014,153.511
C01390=1077.537,-95.852,445.119,173.278,20.013,153.511
C01391=1077.530,-96.102,445.129,173.277,20.012,153.511
C01392=1077.525,-96.351,445.140,173.275,20.010,153.511
C01393=1077.519,-96.601,445.149,173.274,20.009,153.511
C01394=1077.513,-96.851,445.160,173.272,20.008,153.511
C01395=1077.507,-97.101,445.170,173.270,20.007,153.511
C01396=1077.499,-97.381,445.182,173.269,20.005,153.511
C01397=1077.494,-97.661,445.193,173.266,20.003,153.511
C01398=1077.486,-97.941,445.205,173.265,20.002,153.512
C01399=1077.479,-98.221,445.216,173.263,20.001,153.512
C01400=1077.473,-98.471,445.226,173.262,19.999,153.511
C01401=1077.467,-98.721,445.236,173.260,19.998,153.512
C01402=1077.461,-98.970,445.246,173.259,19.997,153.512
C01403=1077.455,-99.220,445.256,173.257,19.995,153.512
C01404=1077.449,-99.470,445.266,173.255,19.994,153.512
C01405=1077.443,-99.719,445.276,173.255,19.993,153.512
C01406=1077.437,-99.969,445.286,173.253,19.993,153.512
C01407=1077.430,-100.219,445.296,173.251,19.991,153.512
C01408=1077.425,-100.468,445.306,173.250,19.990,153.512
C01409=1077.418,-100.719,445.316,173.248,19.989,153.512
C01410=1077.412,-100.968,445.326,173.247,19.987,153.512
C01411=1077.406,-101.218,445.337,173.245,19.986,153.512
C01412=1077.400,-101.468,445.346,173.243,19.985,153.512
C01413=1077.394,-101.717,445.356,173.242,19.984,153.512
C01414=1077.388,-101.967,445.367,173.240,19.982,153.512
C01415=1077.382,-102.217,445.376,173.239,19.981,153.512
C01416=1077.376,-102.467,445.386,173.237,19.980,153.512
C01417=1077.369,-102.716,445.396,173.236,19.979,153.512
C01418=1077.364,-102.966,445.406,173.235,19.978,153.512
C01419=1077.358,-103.216,445.416,173.233,19.977,153.512
C01420=1077.351,-103.465,445.426,173.231,19.976,153.512
C01421=1077.345,-103.715,445.436,173.230,19.975,153.512
C01422=1077.339,-103.965,445.446,173.228,19.973,153.512
C01423=1077.333,-104.214,445.456,173.227,19.972,153.512
C01424=1077.327,-104.464,445.466,173.225,19.971,153.512
C01425=1077.321,-104.713,445.475,173.223,19.970,153.512
C01426=1077.315,-104.964,445.486,173.222,19.968,153.512
C01427=1077.309,-105.213,445.495,173.220,19.967,153.513
C01428=1077.303,-105.463,445.505,173.219,19.966,153.513
C01429=1077.296,-105.712,445.515,173.218,19.966,153.513
C01430=1077.291,-105.962,445.525,173.216,19.964,153.513
C01431=1077.285,-106.212,445.535,173.214,19.963,153.513
C01432=1077.279,-106.462,445.544,173.213,19.962,153.513
C01433=1077.272,-106.711,445.555,173.211,19.961,153.513
C01434=1077.266,-106.961,445.564,173.210,19.960,153.513
C01435=1077.260,-107.211,445.574,173.208,19.958,153.513
C01436=1077.254,-107.461,445.584,173.206,19.957,153.513
C01437=1077.248,-107.711,445.593,173.205,19.956,153.513
C01438=1077.242,-107.960,445.604,173.204,19.955,153.513
C01439=1077.236,-108.210,445.613,173.202,19.955,153.513
C01440=1077.229,-108.459,445.623,173.201,19.953,153.513
C01441=1077.223,-108.709,445.632,173.199,19.952,153.513
C01442=1077.218,-108.959,445.643,173.197,19.951,153.513
C01443=1077.212,-109.209,445.652,173.196,19.950,153.513
C01444=1077.205,-109.458,445.662,173.194,19.949,153.514
C01445=1077.199,-109.708,445.672,173.192,19.948,153.514
C01446=1077.193,-109.958,445.682,173.191,19.946,153.514
C01447=1077.187,-110.208,445.691,173.190,19.946,153.514
C01448=1077.180,-110.458,445.701,173.188,19.945,153.514
C01449=1077.174,-110.707,445.710,173.187,19.944,153.514
C01450=1077.168,-110.957,445.720,173.185,19.943,153.514
C01451=1077.162,-111.207,445.729,173.183,19.942,153.514
C01452=1077.156,-111.457,445.739,173.182,19.940,153.514
C01453=1077.150,-111.707,445.749,173.180,19.939,153.514
C01454=1077.144,-111.957,445.759,173.178,19.938,153.514
C01455=1077.138,-112.206,445.769,173.177,19.938,153.514
C01456=1077.131,-112.456,445.779,173.176,19.936,153.514
C01457=1077.126,-112.705,445.788,173.174,19.935,153.514
C01458=1077.120,-112.955,445.797,173.173,19.935,153.514
C01459=1077.114,-113.204,445.807,173.171,19.934,153.515
C01460=1077.107,-113.483,445.817,173.169,19.932,153.515
C01461=1077.100,-113.759,445.828,173.168,19.931,153.515
C01462=1077.094,-114.036,445.839,173.166,19.930,153.515
C01463=1077.086,-114.314,445.849,173.164,19.929,153.515
C01464=1077.080,-114.564,445.858,173.163,19.928,153.515
C01465=1077.074,-114.814,445.868,173.161,19.927,153.515
C01466=1077.067,-115.064,445.878,173.159,19.926,153.515
C01467=1077.062,-115.313,445.887,173.157,19.925,153.515
C01468=1077.056,-115.563,445.896,173.156,19.924,153.515
C01469=1077.049,-115.812,445.906,173.155,19.923,153.515
C01470=1077.043,-116.062,445.915,173.153,19.922,153.515
C01471=1077.037,-116.312,445.925,173.152,19.921,153.516
C01472=1077.031,-116.562,445.935,173.150,19.920,153.516
C01473=1077.025,-116.812,445.944,173.148,19.919,153.516
C01474=1077.019,-117.061,445.954,173.146,19.918,153.516
C01475=1077.012,-117.311,445.963,173.145,19.917,153.516
C01476=1077.006,-117.561,445.973,173.144,19.917,153.516
C01477=1077.001,-117.810,445.982,173.142,19.916,153.516
C01478=1076.995,-118.060,445.992,173.141,19.915,153.516
C01479=1076.988,-118.310,446.001,173.139,19.914,153.516
C01480=1076.982,-118.560,446.010,173.137,19.913,153.516
C01481=1076.976,-118.810,446.019,173.135,19.912,153.517
C01482=1076.969,-119.059,446.029,173.135,19.911,153.517
C01483=1076.963,-119.309,446.038,173.133,19.910,153.517
C01484=1076.957,-119.559,446.048,173.131,19.910,153.517
C01485=1076.951,-119.808,446.057,173.129,19.909,153.517
C01486=1076.945,-120.058,446.066,173.128,19.908,153.517
C01487=1076.939,-120.308,446.076,173.126,19.906,153.517
C01488=1076.933,-120.558,446.085,173.124,19.905,153.517
C01489=1076.927,-120.808,446.094,173.124,19.905,153.517
C01490=1076.920,-121.057,446.103,173.122,19.904,153.517
C01491=1076.914,-121.307,446.113,173.120,19.903,153.517
C01492=1076.908,-121.556,446.122,173.118,19.902,153.518
C01493=1076.902,-121.806,446.132,173.117,19.901,153.518
C01494=1076.896,-122.057,446.141,173.115,19.900,153.518
C01495=1076.890,-122.306,446.150,173.114,19.900,153.518
C01496=1076.883,-122.556,446.159,173.112,19.899,153.518
C01497=1076.877,-122.806,446.169,173.111,19.898,153.518
C01498=1076.872,-123.055,446.178,173.109,19.897,153.518
C01499=1076.866,-123.305,446.187,173.107,19.896,153.518
C01500=1076.860,-123.555,446.196,173.106,19.895,153.518
C01501=1076.853,-123.805,446.206,173.105,19.895,153.519
C01502=1076.846,-124.054,446.215,173.103,19.894,153.519
C01503=1076.841,-124.304,446.223,173.101,19.893,153.519
C01504=1076.835,-124.554,446.233,173.099,19.892,153.519
C01505=1076.829,-124.804,446.242,173.098,19.891,153.519
C01506=1076.823,-125.053,446.252,173.097,19.891,153.519
C01507=1076.816,-125.303,446.260,173.095,19.890,153.519
C01508=1076.810,-125.553,446.270,173.093,19.889,153.519
C01509=1076.804,-125.802,446.279,173.091,19.888,153.520
C01510=1076.798,-126.052,446.287,173.090,19.887,153.520
C01511=1076.792,-126.302,446.297,173.089,19.887,153.520
C01512=1076.785,-126.552,446.306,173.087,19.886,153.520
C01513=1076.779,-126.802,446.316,173.085,19.885,153.520
C01514=1076.773,-127.051,446.324,173.083,19.884,153.520
C01515=1076.767,-127.301,446.333,173.082,19.884,153.520
C01516=1076.761,-127.551,446.342,173.080,19.883,153.521
C01517=1076.755,-127.801,446.352,173.079,19.882,153.521
C01518=1076.749,-128.052,446.361,173.077,19.881,153.521
C01519=1076.746,-128.302,446.371,173.076,19.879,153.521
C01520=1076.745,-128.557,446.382,173.075,19.877,153.520
C01521=1076.747,-128.810,446.395,173.074,19.874,153.520
C01522=1076.752,-129.064,446.408,173.074,19.869,153.519
C01523=1076.759,-129.314,446.423,173.074,19.864,153.518
C01524=1076.364,-129.337,446.272,173.029,19.991,153.549
C01525=1076.356,-129.085,446.258,173.029,19.996,153.550
C01526=1076.351,-128.832,446.244,173.029,20.001,153.551
C01527=1076.349,-128.579,446.232,173.030,20.004,153.551
C01528=1076.350,-128.325,446.220,173.031,20.007,153.552
C01529=1076.353,-128.074,446.210,173.032,20.009,153.552
C01530=1076.358,-127.824,446.201,173.034,20.010,153.552
C01531=1076.364,-127.573,446.192,173.036,20.011,153.552
C01532=1076.370,-127.323,446.182,173.037,20.012,153.551
C01533=1076.376,-127.073,446.174,173.039,20.012,153.551
C01534=1076.383,-126.824,446.165,173.040,20.012,153.551
C01535=1076.389,-126.574,446.155,173.042,20.013,153.551
C01536=1076.395,-126.324,446.147,173.044,20.014,153.551
C01537=1076.402,-126.074,446.138,173.045,20.015,153.551
C01538=1076.408,-125.825,446.128,173.047,20.016,153.551
C01539=1076.414,-125.575,446.118,173.048,20.017,153.551
C01540=1076.419,-125.325,446.110,173.050,20.017,153.550
C01541=1076.426,-125.076,446.101,173.051,20.018,153.550
C01542=1076.432,-124.826,446.091,173.053,20.019,153.550
C01543=1076.438,-124.575,446.083,173.055,20.020,153.550
C01544=1076.444,-124.325,446.073,173.057,20.021,153.550
C01545=1076.451,-124.077,446.064,173.058,20.021,153.550
C01546=1076.457,-123.827,446.055,173.059,20.022,153.550
C01547=1076.463,-123.577,446.045,173.061,20.023,153.550
C01548=1076.469,-123.327,446.036,173.063,20.024,153.549
C01549=1076.475,-123.077,446.027,173.065,20.025,153.549
C01550=1076.481,-122.828,446.018,173.065,20.025,153.549
C01551=1076.488,-122.578,446.009,173.067,20.026,153.549
C01552=1076.493,-122.328,446.000,173.069,20.027,153.549
C01553=1076.500,-122.078,445.990,173.071,20.028,153.549
C01554=1076.506,-121.828,445.981,173.072,20.029,153.549
C01555=1076.512,-121.578,445.971,173.074,20.030,153.549
C01556=1076.517,-121.329,445.962,173.076,20.031,153.549
C01557=1076.524,-121.080,445.953,173.076,20.032,153.549
C01558=1076.530,-120.830,445.944,173.078,20.033,153.549
C01559=1076.536,-120.580,445.934,173.080,20.034,153.548
C01560=1076.543,-120.330,445.925,173.082,20.035,153.548
C01561=1076.549,-120.080,445.915,173.083,20.035,153.548
C01562=1076.555,-119.830,445.906,173.085,20.036,153.548
C01563=1076.560,-119.581,445.897,173.086,20.037,153.548
C01564=1076.567,-119.331,445.887,173.088,20.038,153.548
C01565=1076.573,-119.081,445.878,173.089,20.039,153.548
C01566=1076.579,-118.832,445.869,173.091,20.040,153.548
C01567=1076.586,-118.582,445.860,173.093,20.041,153.548
C01568=1076.592,-118.332,445.850,173.095,20.041,153.547
C01569=1076.598,-118.082,445.840,173.096,20.043,153.547
C01570=1076.604,-117.832,445.831,173.097,20.043,153.547
C01571=1076.610,-117.583,445.822,173.099,20.044,153.547
C01572=1076.616,-117.333,445.812,173.100,20.045,153.547
C01573=1076.622,-117.084,445.803,173.102,20.046,153.547
C01574=1076.628,-116.834,445.793,173.104,20.047,153.547
C01575=1076.634,-116.584,445.783,173.106,20.048,153.547
C01576=1076.640,-116.334,445.775,173.107,20.049,153.547
C01577=1076.646,-116.084,445.765,173.108,20.050,153.547
C01578=1076.653,-115.834,445.755,173.110,20.051,153.547
C01579=1076.659,-115.584,445.746,173.111,20.052,153.546
C01580=1076.665,-115.334,445.736,173.113,20.053,153.546
C01581=1076.671,-115.086,445.728,173.115,20.054,153.546
C01582=1076.677,-114.836,445.718,173.116,20.055,153.546
C01583=1076.684,-114.586,445.709,173.118,20.056,153.546
C01584=1076.690,-114.336,445.699,173.119,20.057,153.546
C01585=1076.697,-114.059,445.688,173.122,20.058,153.546
C01586=1076.703,-113.781,445.678,173.123,20.059,153.546
C01587=1076.710,-113.503,445.667,173.125,20.060,153.546
C01588=1076.717,-113.227,445.656,173.127,20.061,153.546
C01589=1076.723,-112.977,445.646,173.128,20.063,153.546
C01590=1076.729,-112.727,445.637,173.130,20.064,153.546
C01591=1076.735,-112.477,445.627,173.131,20.064,153.546
C01592=1076.742,-112.227,445.618,173.132,20.066,153.546
C01593=1076.747,-111.977,445.607,173.134,20.066,153.545
C01594=1076.753,-111.727,445.598,173.136,20.067,153.545
C01595=1076.759,-111.478,445.588,173.137,20.068,153.545
C01596=1076.766,-111.228,445.579,173.139,20.070,153.545
C01597=1076.772,-110.978,445.569,173.141,20.071,153.545
C01598=1076.778,-110.728,445.560,173.142,20.072,153.545
C01599=1076.784,-110.478,445.550,173.143,20.073,153.545
C01600=1076.790,-110.229,445.541,173.145,20.074,153.545
C01601=1076.796,-109.980,445.530,173.146,20.074,153.545
C01602=1076.802,-109.730,445.521,173.148,20.076,153.545
C01603=1076.809,-109.481,445.511,173.150,20.077,153.545
C01604=1076.815,-109.231,445.502,173.151,20.078,153.545
C01605=1076.820,-108.981,445.492,173.153,20.079,153.545
C01606=1076.826,-108.731,445.482,173.155,20.080,153.545
C01607=1076.832,-108.481,445.472,173.156,20.081,153.544
C01608=1076.839,-108.232,445.462,173.157,20.082,153.544
C01609=1076.845,-107.982,445.453,173.159,20.083,153.544
C01610=1076.851,-107.732,445.443,173.160,20.084,153.544
C01611=1076.857,-107.483,445.433,173.162,20.085,153.544
C01612=1076.864,-107.233,445.424,173.164,20.086,153.544
C01613=1076.869,-106.983,445.414,173.165,20.088,153.544
C01614=1076.876,-106.733,445.403,173.167,20.089,153.544
C01615=1076.882,-106.484,445.394,173.168,20.090,153.544
C01616=1076.888,-106.234,445.384,173.170,20.091,153.544
C01617=1076.894,-105.984,445.375,173.172,20.093,153.544
C01618=1076.899,-105.734,445.365,173.172,20.093,153.544
C01619=1076.906,-105.485,445.354,173.174,20.095,153.544
C01620=1076.912,-105.235,445.345,173.176,20.095,153.544
C01621=1076.918,-104.985,445.335,173.177,20.097,153.544
C01622=1076.924,-104.735,445.325,173.179,20.098,153.544
C01623=1076.930,-104.486,445.315,173.180,20.099,153.544
C01624=1076.936,-104.236,445.305,173.182,20.100,153.544
C01625=1076.943,-103.986,445.296,173.184,20.102,153.544
C01626=1076.948,-103.736,445.285,173.185,20.103,153.544
C01627=1076.954,-103.487,445.275,173.187,20.104,153.544
C01628=1076.961,-103.237,445.266,173.189,20.105,153.543
C01629=1076.967,-102.987,445.256,173.189,20.106,153.544
C01630=1076.973,-102.737,445.245,173.191,20.107,153.543
C01631=1076.979,-102.487,445.235,173.192,20.108,153.543
C01632=1076.985,-102.238,445.226,173.194,20.109,153.543
C01633=1076.992,-101.988,445.215,173.196,20.111,153.543
C01634=1076.997,-101.738,445.205,173.197,20.112,153.543
C01635=1077.004,-101.488,445.196,173.199,20.113,153.543
C01636=1077.010,-101.239,445.185,173.200,20.115,153.543
C01637=1077.015,-100.989,445.175,173.202,20.116,153.543
C01638=1077.022,-100.739,445.166,173.204,20.117,153.543
C01639=1077.028,-100.490,445.155,173.205,20.118,153.543
C01640=1077.034,-100.240,445.145,173.207,20.119,153.543
C01641=1077.040,-99.990,445.136,173.208,20.121,153.543
C01642=1077.046,-99.741,445.125,173.210,20.122,153.543
C01643=1077.052,-99.491,445.115,173.211,20.123,153.543
C01644=1077.058,-99.242,445.105,173.213,20.124,153.543
C01645=1077.065,-98.991,445.095,173.214,20.125,153.543
C01646=1077.071,-98.742,445.085,173.216,20.127,153.543
C01647=1077.077,-98.492,445.075,173.217,20.128,153.543
C01648=1077.083,-98.242,445.065,173.219,20.129,153.543
C01649=1077.090,-97.962,445.053,173.220,20.131,153.543
C01650=1077.097,-97.682,445.042,173.222,20.131,153.543
C01651=1077.103,-97.401,445.031,173.224,20.133,153.543
C01652=1077.110,-97.121,445.019,173.226,20.135,153.543
C01653=1077.116,-96.871,445.009,173.227,20.136,153.543
C01654=1077.122,-96.622,444.999,173.229,20.137,153.543
C01655=1077.128,-96.372,444.988,173.231,20.139,153.543
C01656=1077.134,-96.123,444.978,173.232,20.140,153.543
C01657=1077.140,-95.873,444.968,173.234,20.142,153.543
C01658=1077.146,-95.624,444.958,173.234,20.143,153.543
C01659=1077.152,-95.373,444.948,173.236,20.144,153.543
C01660=1077.158,-95.124,444.937,173.237,20.145,153.543
C01661=1077.164,-94.873,444.927,173.239,20.147,153.543
C01662=1077.171,-94.624,444.916,173.240,20.148,153.543
C01663=1077.176,-94.374,444.906,173.242,20.149,153.543
C01664=1077.182,-94.125,444.896,173.244,20.150,153.543
C01665=1077.188,-93.875,444.886,173.245,20.152,153.543
C01666=1077.194,-93.626,444.876,173.247,20.153,153.543
C01667=1077.200,-93.376,444.865,173.248,20.155,153.543
C01668=1077.206,-93.126,444.855,173.250,20.156,153.543
C01669=1077.212,-92.876,444.845,173.251,20.157,153.543
C01670=1077.218,-92.626,444.834,173.253,20.159,153.543
C01671=1077.224,-92.377,444.823,173.254,20.160,153.543
C01672=1077.230,-92.127,444.813,173.256,20.162,153.543
C01673=1077.236,-91.878,444.803,173.257,20.163,153.543
C01674=1077.242,-91.628,444.793,173.259,20.164,153.543
C01675=1077.248,-91.378,444.782,173.261,20.165,153.543
C01676=1077.254,-91.129,444.772,173.262,20.167,153.543
C01677=1077.261,-90.878,444.762,173.264,20.168,153.543
C01678=1077.267,-90.629,444.751,173.265,20.170,153.543
C01679=1077.272,-90.379,444.741,173.267,20.171,153.543
C01680=1077.278,-90.130,444.730,173.268,20.173,153.543
C01681=1077.284,-89.880,444.719,173.270,20.174,153.543
C01682=1077.290,-89.630,444.710,173.271,20.175,153.543
C01683=1077.297,-89.380,444.699,173.273,20.177,153.543
C01684=1077.302,-89.131,444.688,173.274,20.178,153.543
C01685=1077.309,-88.881,444.678,173.275,20.179,153.543
C01686=1077.314,-88.631,444.667,173.277,20.180,153.543
C01687=1077.321,-88.382,444.657,173.278,20.182,153.543
C01688=1077.327,-88.131,444.647,173.280,20.183,153.543
C01689=1077.333,-87.882,444.636,173.281,20.185,153.543
C01690=1077.339,-87.633,444.625,173.283,20.186,153.543
C01691=1077.345,-87.383,444.615,173.284,20.188,153.543
C01692=1077.351,-87.133,444.605,173.286,20.189,153.543
C01693=1077.357,-86.883,444.594,173.287,20.190,153.543
C01694=1077.363,-86.634,444.583,173.289,20.192,153.543
C01695=1077.369,-86.384,444.573,173.290,20.193,153.543
C01696=1077.375,-86.134,444.562,173.292,20.195,153.543
C01697=1077.382,-85.885,444.552,173.293,20.196,153.543
C01698=1077.388,-85.635,444.541,173.295,20.198,153.543
C01699=1077.393,-85.385,444.531,173.296,20.199,153.543
C01700=1077.400,-85.136,444.520,173.298,20.200,153.543
C01701=1077.406,-84.886,444.509,173.299,20.202,153.543
C01702=1077.412,-84.636,444.498,173.301,20.203,153.543
C01703=1077.418,-84.387,444.488,173.302,20.205,153.543
C01704=1077.424,-84.137,444.478,173.304,20.206,153.543
C01705=1077.430,-83.887,444.467,173.305,20.208,153.543
C01706=1077.437,-83.637,444.456,173.307,20.209,153.543
C01707=1077.442,-83.388,444.445,173.308,20.211,153.543
C01708=1077.449,-83.138,444.435,173.310,20.212,153.543
C01709=1077.455,-82.888,444.425,173.311,20.214,153.543
C01710=1077.461,-82.638,444.414,173.313,20.215,153.543
C01711=1077.468,-82.389,444.403,173.314,20.217,153.543
C01712=1077.473,-82.139,444.392,173.316,20.218,153.543
C01713=1077.480,-81.861,444.380,173.318,20.219,153.543
C01714=1077.486,-81.583,444.369,173.320,20.221,153.543
C01715=1077.494,-81.305,444.356,173.321,20.223,153.543
C01716=1077.501,-81.028,444.345,173.323,20.224,153.543
C01717=1077.507,-80.778,444.334,173.324,20.226,153.543
C01718=1077.513,-80.528,444.323,173.326,20.227,153.543
C01719=1077.519,-80.278,444.313,173.327,20.229,153.543
C01720=1077.525,-80.029,444.302,173.329,20.230,153.543
C01721=1077.531,-79.778,444.291,173.330,20.232,153.543
C01722=1077.537,-79.529,444.280,173.332,20.234,153.544
C01723=1077.543,-79.279,444.269,173.333,20.235,153.544
C01724=1077.550,-79.030,444.258,173.335,20.237,153.544
C01725=1077.555,-78.780,444.248,173.336,20.238,153.544
C01726=1077.561,-78.531,444.237,173.338,20.239,153.544
C01727=1077.567,-78.280,444.225,173.339,20.241,153.544
C01728=1077.573,-78.031,444.215,173.341,20.242,153.544
C01729=1077.579,-77.781,444.204,173.342,20.244,153.544
C01730=1077.585,-77.532,444.193,173.344,20.246,153.544
C01731=1077.591,-77.282,444.182,173.345,20.247,153.544
C01732=1077.598,-77.033,444.171,173.347,20.249,153.544
C01733=1077.603,-76.783,444.160,173.348,20.250,153.544
C01734=1077.610,-76.533,444.149,173.349,20.252,153.544
C01735=1077.615,-76.283,444.138,173.351,20.254,153.544
C01736=1077.621,-76.034,444.127,173.352,20.255,153.544
C01737=1077.627,-75.784,444.116,173.354,20.257,153.544
C01738=1077.633,-75.534,444.105,173.355,20.258,153.544
C01739=1077.639,-75.284,444.094,173.357,20.260,153.544
C01740=1077.645,-75.035,444.083,173.358,20.262,153.544
C01741=1077.652,-74.785,444.073,173.360,20.263,153.544
C01742=1077.658,-74.535,444.062,173.361,20.264,153.544
C01743=1077.664,-74.286,444.051,173.363,20.266,153.545
C01744=1077.670,-74.036,444.040,173.364,20.268,153.545
C01745=1077.676,-73.786,444.029,173.365,20.269,153.545
C01746=1077.682,-73.536,444.018,173.367,20.271,153.545
C01747=1077.687,-73.287,444.007,173.368,20.273,153.545
C01748=1077.693,-73.036,443.995,173.371,20.275,153.545
C01749=1077.699,-72.788,443.983,173.372,20.276,153.545
C01750=1077.705,-72.538,443.973,173.373,20.278,153.545
C01751=1077.711,-72.288,443.961,173.375,20.280,153.545
C01752=1077.717,-72.038,443.950,173.376,20.281,153.545
C01753=1077.723,-71.789,443.940,173.378,20.283,153.545
C01754=1077.729,-71.539,443.928,173.379,20.285,153.545
C01755=1077.735,-71.289,443.917,173.381,20.286,153.545
C01756=1077.741,-71.040,443.906,173.382,20.288,153.545
C01757=1077.746,-70.790,443.894,173.384,20.290,153.545
C01758=1077.752,-70.540,443.883,173.385,20.291,153.546
C01759=1077.758,-70.291,443.872,173.386,20.293,153.546
C01760=1077.764,-70.041,443.861,173.388,20.294,153.546
C01761=1077.770,-69.791,443.850,173.389,20.296,153.546
C01762=1077.776,-69.542,443.839,173.391,20.298,153.546
C01763=1077.782,-69.292,443.827,173.392,20.299,153.546
C01764=1077.788,-69.043,443.816,173.393,20.301,153.546
C01765=1077.794,-68.792,443.805,173.395,20.303,153.546
C01766=1077.799,-68.543,443.794,173.396,20.305,153.546
C01767=1077.805,-68.294,443.782,173.398,20.306,153.546
C01768=1077.812,-68.044,443.771,173.399,20.308,153.546
C01769=1077.817,-67.794,443.760,173.401,20.310,153.546
C01770=1077.824,-67.544,443.749,173.402,20.311,153.547
C01771=1077.830,-67.295,443.737,173.404,20.314,153.547
C01772=1077.835,-67.045,443.726,173.406,20.315,153.547
C01773=1077.841,-66.795,443.714,173.407,20.317,153.547
C01774=1077.847,-66.546,443.704,173.408,20.319,153.547
C01775=1077.854,-66.296,443.692,173.410,20.320,153.547
C01776=1077.859,-66.047,443.681,173.411,20.322,153.547
C01777=1077.866,-65.771,443.668,173.413,20.324,153.547
C01778=1077.872,-65.495,443.655,173.414,20.326,153.547
C01779=1077.879,-65.219,443.643,173.416,20.328,153.547
C01780=1077.886,-64.943,443.630,173.418,20.329,153.547
C01781=1077.892,-64.693,443.619,173.419,20.331,153.548
C01782=1077.897,-64.444,443.608,173.421,20.333,153.548
C01783=1077.903,-64.194,443.596,173.422,20.335,153.548
C01784=1077.909,-63.945,443.585,173.423,20.336,153.548
C01785=1077.916,-63.695,443.573,173.425,20.338,153.548
C01786=1077.921,-63.446,443.562,173.426,20.340,153.548
C01787=1077.928,-63.195,443.551,173.428,20.341,153.548
C01788=1077.933,-62.946,443.539,173.429,20.343,153.548
C01789=1077.939,-62.696,443.527,173.430,20.345,153.548
C01790=1077.945,-62.446,443.516,173.433,20.347,153.548
C01791=1077.952,-62.197,443.504,173.434,20.349,153.548
C01792=1077.957,-61.947,443.493,173.435,20.351,153.548
C01793=1077.963,-61.698,443.481,173.437,20.352,153.548
C01794=1077.969,-61.448,443.470,173.438,20.354,153.549
C01795=1077.975,-61.198,443.459,173.440,20.356,153.549
C01796=1077.982,-60.949,443.447,173.441,20.358,153.549
C01797=1077.987,-60.698,443.435,173.443,20.359,153.549
C01798=1077.993,-60.450,443.424,173.444,20.361,153.549
C01799=1077.999,-60.199,443.413,173.445,20.362,153.549
C01800=1078.006,-59.951,443.401,173.447,20.364,153.549
C01801=1078.011,-59.700,443.389,173.448,20.366,153.549
C01802=1078.018,-59.450,443.377,173.449,20.368,153.549
C01803=1078.024,-59.201,443.366,173.451,20.369,153.549
C01804=1078.030,-58.951,443.354,173.453,20.372,153.550
C01805=1078.035,-58.702,443.343,173.454,20.374,153.550
C01806=1078.042,-58.452,443.331,173.456,20.375,153.550
C01807=1078.048,-58.203,443.320,173.457,20.377,153.550
C01808=1078.054,-57.953,443.308,173.459,20.379,153.550
C01809=1078.060,-57.702,443.296,173.460,20.381,153.550
C01810=1078.066,-57.454,443.285,173.461,20.382,153.550
C01811=1078.072,-57.203,443.273,173.463,20.384,153.550
C01812=1078.077,-56.954,443.261,173.464,20.386,153.550
C01813=1078.084,-56.704,443.250,173.466,20.388,153.550
